// TIA Portal V16 program export: 4 tag tables, 2 data types, 4 data blocks, 31 code blocks (in call order from the OBs), 84 instance data blocks

VAR_GLOBAL   // PLC tag table "Default tag table"
   "Drive 1 Ready" AT %I0.0 : Bool;   // +MC-21K2:1 - Drive 1 Ready
   "Drive 2 Ready" AT %I0.1 : Bool;   // +MC-21K2:5 - Drive 2 Ready
   "Drive 3 Ready" AT %I0.2 : Bool;   // +MC-21K2:2 - Drive 3 Ready
   "Drive 4 Ready" AT %I0.3 : Bool;   // +MC-21K2:6 - Drive 4 Ready
   "Drive 5 Ready" AT %I0.4 : Bool;   // +MC-21K2:3 - Drive 5 Ready
   "Sensor Trechter" AT %I0.5 : Bool;   // +MC-21K2:7 - Sensor Trechter
   "Sensor Op Band" AT %I0.6 : Bool;   // +MC-21K2:4 Sensor Op Band
   "Sensor Wals (Option)" AT %I0.7 : Bool;   // +MC-21K2:8 - Sensor Wals (Option)
   "ESB Oke" AT %I1.0 : Bool;   // +MC-21K3:1 - ESB Oke
   "ESB Pressend" AT %I1.1 : Bool;   // +MC-21K3:5 - ESB Pressend
   "Reset Active" AT %I1.2 : Bool;   // +MC-21K3:2 - Reset Active
   "Noodsleutel(1)" AT %I1.3 : Bool;   // +MC-21K3:6 - NOODSLEUTEL
   "Alle uitgangen(1)" AT %I1.4 : Bool;   // +MC-21K3:3 - Alle uitgangen
   "Door 1 NC contact" AT %I1.5 : Bool;   // +MC-21K3:7 - Safety Doorswitch 1
   "Door 1 NO contact" AT %I1.6 : Bool;   // +MC-21K3:4 - Safety Doorswitch 1 Normaly open
   "Door 2 NC contact" AT %I1.7 : Bool;   // +MC-21K3:8 - Safety Doorswitch 2
   "Spare(5)" AT %I3.0 : Bool;
   "Spare(6)" AT %I3.1 : Bool;
   "Spare(10)" AT %I180.0 : Bool;   // Spare
   "Spare(11)" AT %I180.1 : Bool;   // Spare
   "Spare(12)" AT %I3.4 : Bool;   // Spare
   "Spare(13)" AT %I3.5 : Bool;   // Spare
   "Spare(14)" AT %I3.6 : Bool;   // Spare
   "Spare(15)" AT %I3.7 : Bool;   // Spare
   "Programma 1" AT %I2.0 : Bool;   // +MC-21K4:1 - Programma 1
   "Programma 2" AT %I2.1 : Bool;   // +MC-21K4:5 - Programma 2 (Option)
   "Programma 3" AT %I2.2 : Bool;   // +MC-21K4:2 - Programma 3
   Cleaning AT %I2.3 : Bool;   // +MC-21K4:6 - Cleaning
   "Start Machine" AT %I2.4 : Bool;   // +MC-21K4:3 - Start Machine
   "Stop Machine" AT %I2.5 : Bool;   // +MC-21K4:7 - Stop Machine
   "Spare(16)" AT %I2.6 : Bool;   // Spare
   Encoder_Z_Puls AT %I2.7 : Bool;   // Spare
   "Safety Relais" AT %Q0.0 : Bool;   // +MC-21K6:1 - Safety Relais
   "Bel Storing" AT %Q0.1 : Bool;   // +MC-21K6:5 - Bel Storing
   Spare AT %Q5.3 : Bool;   // Spare
   "Drive 1 RUN FWD" AT %Q1.0 : Bool;   // +MC-21K8:1 - Drive 1 RUN FWD
   "Drive 1 REV]" AT %Q1.1 : Bool;   // +MC-21K8:5 - Drive 1 REV
   "Drive 1 Speed 1" AT %Q1.2 : Bool;   // +MC-21K8:2 - Drive 1 Speed 1
   "Drive 1 Speed 2" AT %Q1.3 : Bool;   // +MC-21K8:6 - Drive 1 Speed 2
   "Spare(3)" AT %Q1.4 : Bool;   // Spare
   "Drive 2 RUN FWD" AT %Q1.5 : Bool;   // +MC-21K8:7 - Drive 2 RUN FWD
   "Drive 2 REV" AT %Q1.6 : Bool;   // +MC-21K8:4 - Drive 2 REV
   "Drive 2 Speed 1" AT %Q1.7 : Bool;   // +MC-21K8:8 - Drive 2 Speed 1
   "Drive 2 Speed 2" AT %Q2.0 : Bool;   // +MC-21K9:1 - Drive 2 Speed 2
   "Spare(4)" AT %Q2.1 : Bool;   // Spare
   "Drive 3 RUN FWD" AT %Q2.2 : Bool;   // +MC-21K9:2 - Drive 3 RUN FWD
   "Drive 3 REV" AT %Q2.3 : Bool;   // +MC-21K9:6 - Drive 3 REV
   "Drive 3 Speed 1" AT %Q2.4 : Bool;   // +MC-21K9:3 - Drive 3 Speed 1
   "Drive 3 Speed 2" AT %Q2.5 : Bool;   // +MC-21K9:7 - Drive 3 Speed 2
   "Spare(21)" AT %Q2.6 : Bool;   // Spare
   "Drive 4 RUN FWD" AT %Q2.7 : Bool;   // +MC-21K9:8 - Drive 4 RUN FWD
   "Drive 4 REV" AT %Q3.0 : Bool;   // +MC-21K10:1 - Drive 4 REV
   "Drive 4 Speed 1" AT %Q3.1 : Bool;   // +MC-21K10:5 - Drive 4 Speed 1
   "Drive 4 Speed 2" AT %Q3.2 : Bool;   // +MC-21K10:2 - Drive 4 Speed 2
   "Spare(22)" AT %Q3.3 : Bool;   // Spare
   "Drive 5 RUN FWD" AT %Q3.4 : Bool;   // +MC-21K10:3 - Drive 5 RUN FWD
   "Drive 5 REV" AT %Q3.5 : Bool;   // +MC-21K10:7 - Drive 5 REV
   "Drive 5 Speed 1" AT %Q3.6 : Bool;   // +MC-21K10:4 - Drive 5 Speed 1
   "Drive 5 Speed 2" AT %Q3.7 : Bool;   // +MC-21K10:8 - Drive 5 Speed 2
   "Spare(23)" AT %Q4.0 : Bool;   // Spare
   "LED Programma 1" AT %Q4.1 : Bool;   // +MC-21K11:5 - LED Programma 1
   "LED Programma 2" AT %Q4.2 : Bool;   // +MC-21K11:2 - LED Programma 2
   "LED Programma 3" AT %Q4.3 : Bool;   // +MC-21K11:6 - LED Programma 3
   "LED E-STOP" AT %Q0.2 : Bool;   // +MC-21K6:2- LED E-STOP
   "LED RUN" AT %Q4.5 : Bool;   // +MC-21K11:7 - LED RUN
   "Valve 1" AT %Q4.6 : Bool;   // +MC-21K11:4 - Valve 1
   "Valve 2" AT %Q4.7 : Bool;   // +MC-21K11:8 - Valve 2
   "Valve 3" AT %Q5.0 : Bool;   // +MC-21K12:1 - Valve 3
   "Valve 4" AT %Q5.1 : Bool;   // +MC-21K12:5 - Valve 4
   "Valve 5" AT %Q5.2 : Bool;   // +MC-21K12:2 - Valve 5
   "Spare(1)" AT %Q6.0 : Bool;   // Spare
   "Spare(2)" AT %Q6.1 : Bool;   // Spare
   "Spare(18)" AT %Q6.2 : Bool;   // Spare
   "Spare(19)" AT %Q6.3 : Bool;   // Spare
   "Spare(20)" AT %Q4.4 : Bool;   // Spare
   "Drive 1 Rapid Stop" AT %Q0.3 : Bool;   // +MC-21K6:6 - Drive 1 Rapid Stop
   "Drive 2 Rapid Stop" AT %Q0.4 : Bool;   // +MC-21K6:3 - Drive 2 Rapid Stop
   "Drive 3 Rapid Stop" AT %Q0.5 : Bool;   // +MC-21K6:7 - Drive 3 Rapid Stop
   "Drive 4 Rapid Stop" AT %Q0.6 : Bool;   // +MC-21K6:4 - Drive 4 Rapid Stop
   "Drive 5 Rapid Stop" AT %Q0.7 : Bool;   // +MC-21K6:8 - Drive 5 Rapid Stop
   "Systeem RUN" AT %M0.0 : Bool;   // Systeem RUN
   Tag_1 AT %M0.1 : Bool;
   Tag_2 AT %M0.2 : Bool;
   Tag_3 AT %M0.3 : Bool;
   Tag_4 AT %M0.4 : Bool;
   "Safety Feedback" AT %M0.6 : Bool;
   Tag_5 AT %M0.7 : Bool;
   Tag_6 AT %M1.0 : Bool;
   "ONC Drive 1 RUN FWD" AT %M10.0 : Bool;
   "ONC Drive 2 RUN FWD" AT %M10.1 : Bool;
   "ONC Drive 3 RUN FWD" AT %M10.2 : Bool;
   "ONC Drive 4 RUN FWD" AT %M10.3 : Bool;
   "ONC Drive 5 RUN FWD" AT %M10.4 : Bool;
   "ONC Drive 1 RUN FWD and Speed 1" AT %M10.5 : Bool;
   "ONC Drive 2 RUN FWD and Speed 1" AT %M10.6 : Bool;
   "ONC Drive 3 RUN FWD and Speed 1" AT %M10.7 : Bool;
   "ONC Drive 4 RUN FWD and Speed 1" AT %M11.0 : Bool;
   "ONC Drive 5 RUN FWD and Speed 1" AT %M11.1 : Bool;
   "ONC Drive 1 RUN FWD and Speed 2" AT %M11.2 : Bool;
   "ONC Drive 2 RUN FWD and Speed 2" AT %M11.3 : Bool;
   "ONC Drive 3 RUN FWD and Speed 2" AT %M11.4 : Bool;
   "ONC Drive 4 RUN FWD and Speed 2" AT %M11.5 : Bool;
   "ONC Drive 5 RUN FWD and Speed 2" AT %M11.6 : Bool;
   Startknop_Scherm AT %M15.0 : Bool;
   Stopknop_Scherm AT %M15.1 : Bool;
   Tag_7 AT %M110.1 : Bool;
   Reset_scherm AT %M15.2 : Bool;
   Sensor_op_band_memory AT %M15.3 : Bool;
   "System RUN_1" AT %M20.0 : Bool;
   ResetDelay AT %M20.1 : Bool;
   SensorWalsMemory AT %M20.2 : Bool;
   Timer_Memory AT %M20.3 : Bool;
   StopAll AT %M20.4 : Bool;
   Tag_8 AT %M100.3 : Bool;
   Tag_9 AT %M100.4 : Bool;
   Tag_10 AT %M0.5 : Bool;
   Tag_11 AT %M150.0 : Bool;
   Tag_12 AT %M101.1 : Bool;
   Tag_13 AT %T1 : Timer;
   Tag_14 AT %M300.0 : Bool;
   Tag_15 AT %M260.0 : Bool;
   Tag_16 AT %M300.1 : Bool;
   Tag_17 AT %M501.0 : Bool;
   Tag_18 AT %M500.1 : Bool;
   Tag_19 AT %M160.0 : Bool;
   Tag_20 AT %M150.5 : Bool;
   Tag_21 AT %QD256 : DWord;
   Tag_22 AT %QW260 : Word;
   Tag_23 AT %ID256 : DWord;
   Tag_24 AT %ID260 : DWord;
   Tag_25 AT %ID464 : DWord;
   Tag_26 AT %ID471 : DWord;
   Tag_27 AT %QW471 : Word;
   Tag_28 AT %QD464 : DWord;
   Tag_30 AT %IW205 : Int;
   SystemTime AT %MD2 : Time;
   Tag_31 AT %M5.0 : Bool;
   Lamp_Green AT %Q7.0 : Bool;
   Lamp_Blue AT %Q7.1 : Bool;
   Lamp_Yellow AT %Q7.2 : Bool;
   Lamp_Red AT %Q7.3 : Bool;
   Lamp_Buzzer AT %Q7.4 : Bool;
   PulseTimer AT %T0 : Timer;
END_VAR

VAR_GLOBAL   // PLC tag table "PositionControl"
   Counter1_IW100 AT %IW100 : Int;
   Counter2_IW102 AT %IW102 : Int;
   "Manual Jog Fwd" AT %M137.0 : Bool;
   "Manual Jog Rev" AT %M137.1 : Bool;
   ReferenceSwitchAxis3 AT %I3.0 : Bool;
   EncoderBand_Alive AT %IW110 : Int;
   EncoderBand_RawCounter AT %IW112 : Int;
   EncoderBand_FineCounter AT %IW113 : Int;
   Zpuls_Encoder_Band AT %I110.3 : Bool;
END_VAR

VAR_GLOBAL   // PLC tag table "Secund. Tags"
   Aanvoerband_Tag1 AT %M100.0 : Bool;
   Aanvoerband_Tag2 AT %M100.1 : Bool;
   Trechter_Bijvullen_Haltveroorzaker AT %M100.2 : Bool;
   Safety_Automatic AT %M100.5 : Bool;
   Safety_Override AT %M100.6 : Bool;
   RUN_Automatic AT %M100.7 : Bool;
   RUN_Manual AT %M101.0 : Bool;
   Invert_Trechter_Sensor AT %M101.2 : Bool;
   WalsSensorMemory AT %M101.3 : Bool;
   Disable_Module AT %M101.4 : Bool;
   Sensor_Trechter_Delayed AT %M101.5 : Bool;
   Positive_Flank AT %M101.6 : Bool;
   ProductSensor_Flank AT %M101.7 : Bool;
   ProductSensor_Rug AT %M102.0 : Bool;
   SensorRug AT %M102.1 : Bool;
   TimeCyclusEnd AT %M102.2 : Bool;
   CounterReset AT %M102.3 : Bool;
   StartTimer AT %M102.4 : Bool;
   StopTimer AT %M102.5 : Bool;
   SaveTimervalue AT %M102.6 : Bool;
   ResetTotalProducts AT %M102.7 : Bool;
   MaintenanceNeeded AT %M103.0 : Bool;
   RetainValues AT %M112.0 : Bool;
   "Retain_1_DontTouch!" AT %M112.1 : Bool;
   Safety_Doors AT %M112.2 : Bool;
   Overname_Linked_Drive1 AT %M112.3 : Bool;
   Drive_RefuseLinkingDrive1 AT %M112.4 : Bool;
   Drive_4_Speed1_Link AT %M112.5 : Bool;
   Drive_4_Speed1_Unlink AT %M112.6 : Bool;
   SafetyOK AT %M112.7 : Bool;
   Valve2_Pulse AT %M113.0 : Bool;
END_VAR

VAR_GLOBAL   // PLC tag table "Tag table_1"
END_VAR

TYPE "ProductEntry"
// stored: IsFailsafeCompliant false
   STRUCT
      StartTime : Time := T#0ms;
      Active : Bool;
   END_STRUCT;
END_TYPE

TYPE "ProductTrack"
// stored: IsFailsafeCompliant false
   STRUCT
      StartPosition : Real;
      Active : Bool;
   END_STRUCT;
END_TYPE

DATA_BLOCK "PLCMemory"   // DB15
VERSION : 0.1
// stored: AutoNumber true, IsOnlyStoredInLoadMemory false, IsWriteProtectedInAS false
   VAR RETAIN
      Homing_Sensor_Wals_Offset_Test : Time := T#1S_200MS;   // Offset of homing position sensor wals
      Wals_Delay_Offset : Time := T#400MS;   // Offset of Wals on delay
      Safety_Delay : Time := T#5MS;   // Delay of safety high
      WalsCheck_Time : Time := T#5S;   // Time offset when wals slipping message is displayed
      ProductCheck_Time : Time := T#15S;   // Time offset when aanvoer not in position message is displayed
      ProductIntervalTime : Time;   // Counts the time between 2 products
      ProductIntervalTime_1 : Time;   // Depends on ProductIntervalTimer
      ProductIntervalTime_2 : Time;   // Depends on ProductIntervalTimer_1
      TD_Products_Counter : Int;   // Counts the total amount of products with the Sensor Band
      UsernameMemory : String := 'Key';
      PasswordMemory : String := 'Key123';
      SpeedSettingsTakeover : Bool := True;   // Makes the speed of Overname the same as speed Drive 1
      SpeedSettingOvername : Bool;   // Parameter of setting the speed for Drive 4 (Overname)
      SpeedSettingBand : Bool;   // Parameter of setting the speed for Drive 1 (Band)
      TimingSettingOvername : Bool := True;   // Makes the timing of Overname the same as speed Drive 1
      EncoderPosition : Real;   // Real Value of Encoder Axis 3 (Wals)
      StepSize : Real := 0.0;   // Pulsfactor of Encoder Axis 3
      Desired_Encoder_Position : Real;
      Tolerance : Real := 0.0;
      "Encoder PulsOffset" : Time := T#3MS;
      Axis3_Ref_Pos : Real := 85.0;   // Refention position of Axis 3 without tolerance
      Reference_Position_Axis3 : Real;   // Refention position of Axis 3 with calculated tolerance
      ProductCount : Int;
      Axis3_ControlMode : Bool := true;
      Axis1_ControlMode : Bool := true;
      ProductsToProduce : Int;
      SystemTime : Time;
      Disable_Modules : Struct
         Disable_Band : Bool;
         Disable_Trilgoten : Bool;
         Disable_AanvoerWals : Bool;
         Disable_Aandruk1 : Bool;
         Disable_Aandruk2 : Bool;
         Disable_Aandruk3 : Bool;
         Disable_Blaaspuls : Bool;
         Disable_Retourband : Bool;
         Disable_Afsluiter : Bool;
      END_STRUCT;
      Offset_Timers : Struct
         Trilgoten_Start_Offset : Time := T#10MS;   // Delay offset of start trilgoten
         Trilgoten_Stop_Offset : Time := T#10MS;   // Delay offset of stop trilgoten
         Aanvoer_Start_Offset : Time := T#10MS;   // Delay offset of start aanvoer
         Magazijn_Sensor_Delay : Time := T#15S;   // Delay on magazijn sensor.
         Aanvoer_Stop_Offset : Time := T#10MS;   // Delay offset of stop aanvoer
         Overname_Start_Offset : Time := T#5MS;   // Delay offset of start Overname
         Overname_Stop_Offset : Time := T#5MS;   // Delay offset of stop Overname
         Retourband_Start_Offset : Time := T#5ms;
         Retourband_Stop_Offset : Time := T#5ms;
         BlowOff_CycleTime : Time := T#500ms;
         Blow_Off_PulseTime : Time := T#500ms;
      END_STRUCT;
      ProductBuffer : Struct
         DelayTime : Time := T#7s;
         ProductsCount : Int;
         MoveTrigger : Bool;
         MoveFeedback : Bool;
         RestFeedback : Bool;
         InsertIndex : Int;
      END_STRUCT;
      ProductBufferBehindWals : Struct
         DelayTime : Time := T#2s_500MS;
         Product_Count : Int;
      END_STRUCT;
   END_VAR
BEGIN
END_DATA_BLOCK

DATA_BLOCK "DB_SystemTimeCounter"   // DB68
VERSION : 0.1
// stored: AutoNumber true, IsOnlyStoredInLoadMemory false, IsWriteProtectedInAS false
   VAR RETAIN
      SystemTime : Time;
   END_VAR
BEGIN
END_DATA_BLOCK

DATA_BLOCK "Alarms"   // DB24
VERSION : 0.1
// stored: AutoNumber true, IsOnlyStoredInLoadMemory false, IsWriteProtectedInAS false
   VAR
      AlarmStruct : Struct
         Alarm_Product_Not_Position : Bool;
         Alarm_Axis_Not_Position : Bool;
         Alarm_Drive1 : Bool;
         Alarm_Drive2 : Bool;
         Alarm_Drive3 : Bool;
         Alarm_Drive4 : Bool;
         Alarm_Drive5 : Bool;
         "Alarm_To_Many_Products_Reset_Counter!" : Bool;
      END_STRUCT;
      AlarmsWord : Word;
      HMI_Alarm_Drive1 : Word;
      HMI_Alarm_Drive2 : Word;
      HMI_Alarm_Drive3 : Word;
      HMI_Alarm_Drive4 : Word;
      HMI_Alarm_Drive5 : Word;
   END_VAR
BEGIN
END_DATA_BLOCK

DATA_BLOCK "PositionManagement"   // DB51
VERSION : 0.1
// stored: AutoNumber true, IsOnlyStoredInLoadMemory false, IsWriteProtectedInAS false
   VAR RETAIN
      Data : Struct   // Data
         CntPlsPrev : DInt := 0;   // Flowpulsen vorige scan
         CntPlsDiff : DInt := 0;   // Flowpulsen verschil
         CntPlsAct : DInt := 0;   // Flowpulsen actueel
         DosActueel : Real := 0.0;   // Dosering actueel ('x' gram/liter/kg gist)
         Actual_Axis3_Position : Real;   // Actual Position of Axis 3 stored in this datablock
         Actual_Axis1_Position : Real;
      END_STRUCT;
      "Axis 3" : Struct
         Values : Struct
            AxisName : String := 'Drive 3 - Wals';
            "Reference Position" : Int := 0;
            "Set Position" : Real := -50.0;
            "Rest Position" : Real := -25.0;
            Acceleration : Real := 0.0;
            Deacceleration : Real;
            "Axis Correction" : Real := 1.0E-06;
            "Position Offset" : Real := 35.0;
            Pulsfactor : Real := 0.82;
            Axis_Speed : Int := 0;
         END_STRUCT;
         Commands : Struct
            "Go To Rest" : Bool;
            "Start Ref Run" : Bool;
            "Take Over Pos" : Bool;
            "Go To Position" : Bool;
            "Jog Fwd" : Bool;
            "Jog Rev" : Bool;
            Axis_Brake : Bool;
            MasterWord : String;
            "Master Callback" : String;
         END_STRUCT;
         Messages : Struct
            "Axis Busy" : Bool;
            "Error Executing Command" : Bool;
            "Axis On Rest" : Bool;
            "Axis On Position" : Bool;
            "Drive State (Option)" : String;
            "Slip State" : String;
            AxisHasReference : Bool;
         END_STRUCT;
      END_STRUCT;
      Demo_Pos : Struct
         Desired_Pos : Real;
         Start : Bool;
         SetRefRunActive : Bool;
         RequestMove1 : Bool;
         RequestMove2 : Bool;
         PositionMove2 : Real := -330.0;
         PositionMove1 : Real := -120.0;
         Pos2Done : Bool;
         BrakeOnPos1 : Bool;
         BrakeOnPos2 : Bool;
         ManualSensorOverride : Bool;
      END_STRUCT;
      Axis_1 : Struct
         Values : Struct
            AxisName : String := 'Drive 1 - Infeed';
            "Reference Position" : Int := 0;
            "Set Position" : Real := 0.0;
            "Rest Position" : Real := 0.0;
            Acceleration : Real := 0.0;
            Deacceleration : Real;
            "Axis Correction" : Real := 1.0E-06;
            "Position Offset" : Real := 0.001;
            Pulsfactor : Real := -0.325;
            Axis_Speed : Int := 0;
         END_STRUCT;
         Commands : Struct
            "Go To Rest" : Bool;
            "Start Ref Run" : Bool;
            "Take Over Pos" : Bool;
            "Go To Position" : Bool;
            "Jog Fwd" : Bool;
            "Jog Rev" : Bool;
            Axis_Brake : Bool;
            ReferenceSwitch : Bool;
            MasterWord : String;
            "Master Callback" : String;
         END_STRUCT;
         Messages : Struct
            "Axis Busy" : Bool;
            "Error Executing Command" : Bool;
            "Axis On Rest" : Bool;
            "Axis On Position" : Bool;
            "Drive State (Option)" : String;
            "Slip State" : String;
            AxisHasReference : Bool;
         END_STRUCT;
      END_STRUCT;
   END_VAR
BEGIN
END_DATA_BLOCK

ORGANIZATION_BLOCK "OB1"   // OB1, LAD, ProgramCycle
TITLE = MAIN Program
VERSION : 0.1
// MAIN Block
// stored: IsIECCheckEnabled false
   VAR_TEMP
      Temp_0 : Byte;
      Temp_1 : Byte;
      Temp_2 : Byte;
      Temp_3 : Byte;
      Temp_4 : Byte;
      Temp_5 : Byte;
      Temp_6 : Int;
      Temp_7 : Int;
      Temp_8 : Int;
      Temp_9 : Date_And_Time;
      Temp_10 : DWord;
      EncoderDirection : Bool;
      HomingActive : Bool;
      EncError : Bool;
      SafetyActive : Bool;
      "Spare Drive 6" : Bool;
      "Spare Drive 7" : Bool;
      "Spare Drive 8" : Bool;
      "Spare Drive 9" : Bool;
      "Spare Drive 10" : Bool;
      SAFE_OK_Signal : Bool;
      Raw_Position : Real;
      Encoder : Int;
      Gate : Bool;
      GATESTP : Bool;
      OTERRA : Bool;
      Direct : Bool;
      Prepar : Bool;
      CMPV1 : Bool;
      CMPV2 : Bool;
      RESSYNC : Bool;
      RESZERO : Bool;
      OTERR : Bool;
      UnscPos : Int;
      Sc_Pos : Int;
      ActEncPos : Real;
      Start_ReferenceRun : Bool;
      ReferenceSwitch_Input : Bool;
      "Reference Position" : Real;
      "Jog FWD" : Bool;
      "Jog REV" : Bool;
      RefSwitchTemp : Bool;
      RefPosDint : DInt;
      RefPosInt : Real;
      Start_Movement : Bool;
      ClockTime : Int;
      LT_Time : Date_And_Time;
      Summer : Bool;
      SystemStartUp : Bool;
      StartupLow : Bool;
      ManualSensorOverride : Bool;
      Axis1_ScaledPosition : Real;
      Axis1_ActualEncPosition : Real;
   END_VAR
   VAR_TEMP   // added for the SCL form of the ladder/FBD networks
      _w1 : Bool;
   END_VAR
BEGIN

REGION Network 1: Retain Variables
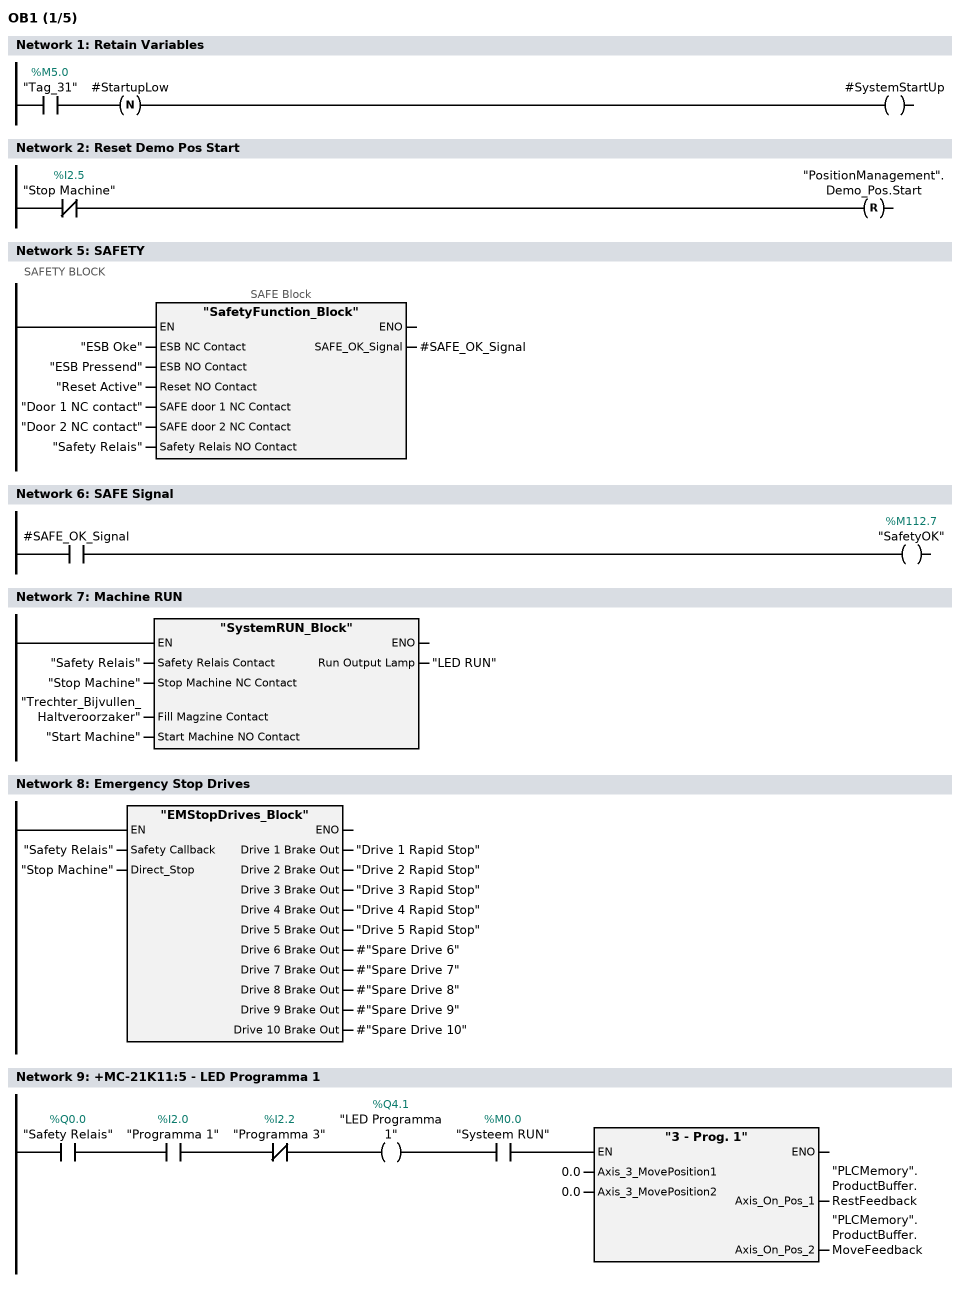
   RUNG wire#powerrail
      Contact( "Tag_31" )
      N_Trig( #StartupLow )
      Coil( #SystemStartUp )
   END_RUNG
   // the same network as SCL:
   #_w1 := NOT "Tag_31" AND #StartupLow;   // falling edge
   #StartupLow := "Tag_31";
   #SystemStartUp := #_w1;
END_REGION

REGION Network 2: Reset Demo Pos Start
   RUNG wire#powerrail
      I_Contact( "Stop Machine" )
      R_Coil( "PositionManagement".Demo_Pos.Start )
   END_RUNG
   // the same network as SCL:
   IF NOT "Stop Machine" THEN "PositionManagement".Demo_Pos.Start := FALSE; END_IF;
END_REGION

REGION Network 3: Retain Veriables (2)
END_REGION

REGION Network 4: System Time
END_REGION

REGION Network 5: SAFETY
   // SAFETY BLOCK
   RUNG wire#powerrail
      "SafetyFunction_Block"("ESB NC Contact" := "ESB Oke", "ESB NO Contact" := "ESB Pressend", "Reset NO Contact" := "Reset Active", "SAFE door 1 NC Contact" := "Door 1 NC contact", "SAFE door 2 NC Contact" := "Door 2 NC contact", "Safety Relais NO Contact" := "Safety Relais", SAFE_OK_Signal => #SAFE_OK_Signal)   // SAFE Block
   END_RUNG
   // the same network as SCL:
   "SafetyFunction_Block"("ESB NC Contact" := "ESB Oke",   // SAFE Block
                          "ESB NO Contact" := "ESB Pressend",
                          "Reset NO Contact" := "Reset Active",
                          "SAFE door 1 NC Contact" := "Door 1 NC contact",
                          "SAFE door 2 NC Contact" := "Door 2 NC contact",
                          "Safety Relais NO Contact" := "Safety Relais",
                          SAFE_OK_Signal => #SAFE_OK_Signal);
END_REGION

REGION Network 6: SAFE Signal
   RUNG wire#powerrail
      Contact( #SAFE_OK_Signal )
      Coil( "SafetyOK" )
   END_RUNG
   // the same network as SCL:
   "SafetyOK" := #SAFE_OK_Signal;
END_REGION

REGION Network 7: Machine RUN
   RUNG wire#powerrail
      "SystemRUN_Block"("Safety Relais Contact" := "Safety Relais", "Stop Machine NC Contact" := "Stop Machine", "Fill Magzine Contact" := "Trechter_Bijvullen_Haltveroorzaker", "Start Machine NO Contact" := "Start Machine", "Run Output Lamp" => "LED RUN")
   END_RUNG
   // the same network as SCL:
   "SystemRUN_Block"("Safety Relais Contact" := "Safety Relais",
                     "Stop Machine NC Contact" := "Stop Machine",
                     "Fill Magzine Contact" := "Trechter_Bijvullen_Haltveroorzaker",
                     "Start Machine NO Contact" := "Start Machine",
                     "Run Output Lamp" => "LED RUN");
END_REGION

REGION Network 8: Emergency Stop Drives
   RUNG wire#powerrail
      "EMStopDrives_Block"("Safety Callback" := "Safety Relais", Direct_Stop := "Stop Machine", "Drive 1 Brake Out" => "Drive 1 Rapid Stop", "Drive 2 Brake Out" => "Drive 2 Rapid Stop", "Drive 3 Brake Out" => "Drive 3 Rapid Stop", "Drive 4 Brake Out" => "Drive 4 Rapid Stop", "Drive 5 Brake Out" => "Drive 5 Rapid Stop", "Drive 6 Brake Out" => #"Spare Drive 6", "Drive 7 Brake Out" => #"Spare Drive 7", "Drive 8 Brake Out" => #"Spare Drive 8", "Drive 9 Brake Out" => #"Spare Drive 9", "Drive 10 Brake Out" => #"Spare Drive 10")
   END_RUNG
   // the same network as SCL:
   "EMStopDrives_Block"("Safety Callback" := "Safety Relais",
                        Direct_Stop := "Stop Machine",
                        "Drive 1 Brake Out" => "Drive 1 Rapid Stop",
                        "Drive 2 Brake Out" => "Drive 2 Rapid Stop",
                        "Drive 3 Brake Out" => "Drive 3 Rapid Stop",
                        "Drive 4 Brake Out" => "Drive 4 Rapid Stop",
                        "Drive 5 Brake Out" => "Drive 5 Rapid Stop",
                        "Drive 6 Brake Out" => #"Spare Drive 6",
                        "Drive 7 Brake Out" => #"Spare Drive 7",
                        "Drive 8 Brake Out" => #"Spare Drive 8",
                        "Drive 9 Brake Out" => #"Spare Drive 9",
                        "Drive 10 Brake Out" => #"Spare Drive 10");
END_REGION

REGION Network 9: +MC-21K11:5 - LED Programma 1
   RUNG wire#powerrail
      Contact( "Safety Relais" )
      Contact( "Programma 1" )
      I_Contact( "Programma 3" )
      Coil( "LED Programma 1" )
      Contact( "Systeem RUN" )
      "3 - Prog. 1"(Axis_3_MovePosition1 := 0.0, Axis_3_MovePosition2 := 0.0, Axis_On_Pos_1 => "PLCMemory".ProductBuffer.RestFeedback, Axis_On_Pos_2 => "PLCMemory".ProductBuffer.MoveFeedback)
   END_RUNG
   // the same network as SCL:
   "LED Programma 1" := "Safety Relais" AND "Programma 1" AND NOT "Programma 3";
   IF "LED Programma 1" AND "Systeem RUN" THEN
       "3 - Prog. 1"(Axis_3_MovePosition1 := 0.0,
                     Axis_3_MovePosition2 := 0.0,
                     Axis_On_Pos_1 => "PLCMemory".ProductBuffer.RestFeedback,
                     Axis_On_Pos_2 => "PLCMemory".ProductBuffer.MoveFeedback);
   END_IF;
END_REGION

REGION Network 10: +MC-21K11:2 - LED Programma 2
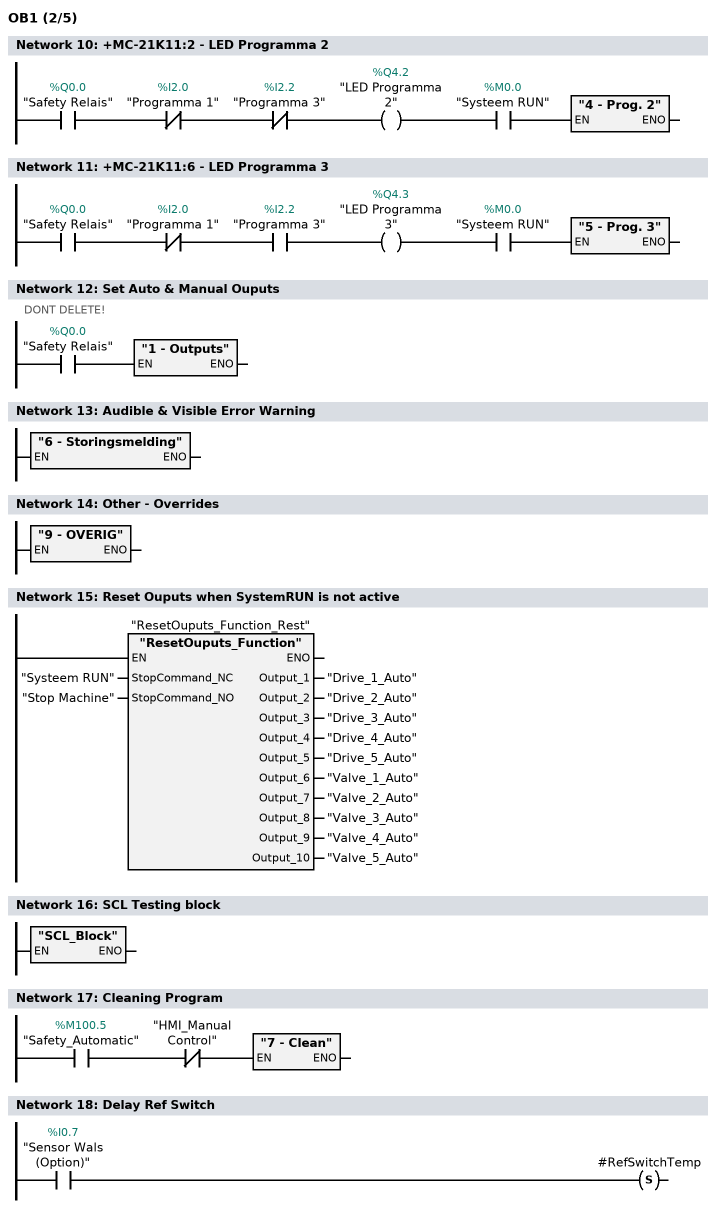
   RUNG wire#powerrail
      Contact( "Safety Relais" )
      I_Contact( "Programma 1" )
      I_Contact( "Programma 3" )
      Coil( "LED Programma 2" )
      Contact( "Systeem RUN" )
      "4 - Prog. 2"()
   END_RUNG
   // the same network as SCL:
   "LED Programma 2" := "Safety Relais" AND NOT "Programma 1" AND NOT "Programma 3";
   IF "LED Programma 2" AND "Systeem RUN" THEN "4 - Prog. 2"(); END_IF;
END_REGION

REGION Network 11: +MC-21K11:6 - LED Programma 3
   RUNG wire#powerrail
      Contact( "Safety Relais" )
      I_Contact( "Programma 1" )
      Contact( "Programma 3" )
      Coil( "LED Programma 3" )
      Contact( "Systeem RUN" )
      "5 - Prog. 3"()
   END_RUNG
   // the same network as SCL:
   "LED Programma 3" := "Safety Relais" AND NOT "Programma 1" AND "Programma 3";
   IF "LED Programma 3" AND "Systeem RUN" THEN "5 - Prog. 3"(); END_IF;
END_REGION

REGION Network 12: Set Auto & Manual Ouputs
   // DONT DELETE!
   RUNG wire#powerrail
      Contact( "Safety Relais" )
      "1 - Outputs"()
   END_RUNG
   // the same network as SCL:
   IF "Safety Relais" THEN "1 - Outputs"(); END_IF;
END_REGION

REGION Network 13: Audible & Visible Error Warning
   RUNG wire#powerrail
      "6 - Storingsmelding"()
   END_RUNG
   // the same network as SCL:
   "6 - Storingsmelding"();
END_REGION

REGION Network 14: Other - Overrides
   RUNG wire#powerrail
      "9 - OVERIG"()
   END_RUNG
   // the same network as SCL:
   "9 - OVERIG"();
END_REGION

REGION Network 15: Reset Ouputs when SystemRUN is not active
   RUNG wire#powerrail
      "ResetOuputs_Function_Rest"(StopCommand_NC := "Systeem RUN", StopCommand_NO := "Stop Machine", Output_1 => "Drive_1_Auto", Output_2 => "Drive_2_Auto", Output_3 => "Drive_3_Auto", Output_4 => "Drive_4_Auto", Output_5 => "Drive_5_Auto", Output_6 => "Valve_1_Auto", Output_7 => "Valve_2_Auto", Output_8 => "Valve_3_Auto", Output_9 => "Valve_4_Auto", Output_10 => "Valve_5_Auto")
   END_RUNG
   // the same network as SCL:
   "ResetOuputs_Function_Rest"(StopCommand_NC := "Systeem RUN",   // "ResetOuputs_Function"
                           StopCommand_NO := "Stop Machine",
                           Output_1 => "Drive_1_Auto",
                           Output_2 => "Drive_2_Auto",
                           Output_3 => "Drive_3_Auto",
                           Output_4 => "Drive_4_Auto",
                           Output_5 => "Drive_5_Auto",
                           Output_6 => "Valve_1_Auto",
                           Output_7 => "Valve_2_Auto",
                           Output_8 => "Valve_3_Auto",
                           Output_9 => "Valve_4_Auto",
                           Output_10 => "Valve_5_Auto");
END_REGION

REGION Network 16: SCL Testing block
   RUNG wire#powerrail
      "SCL_Block"()
   END_RUNG
   // the same network as SCL:
   "SCL_Block"();
END_REGION

REGION Network 17: Cleaning Program
   RUNG wire#powerrail
      Contact( "Safety_Automatic" )
      I_Contact( "HMI_ManualControl" )
      "7 - Clean"()
   END_RUNG
   // the same network as SCL:
   IF "Safety_Automatic" AND NOT "HMI_ManualControl" THEN "7 - Clean"(); END_IF;
END_REGION

REGION Network 18: Delay Ref Switch
   RUNG wire#powerrail
      Contact( "Sensor Wals (Option)" )
      S_Coil( #RefSwitchTemp )
   END_RUNG
   // the same network as SCL:
   IF "Sensor Wals (Option)" THEN #RefSwitchTemp := TRUE; END_IF;
END_REGION

REGION Network 19: Reset Ref Switch Temp
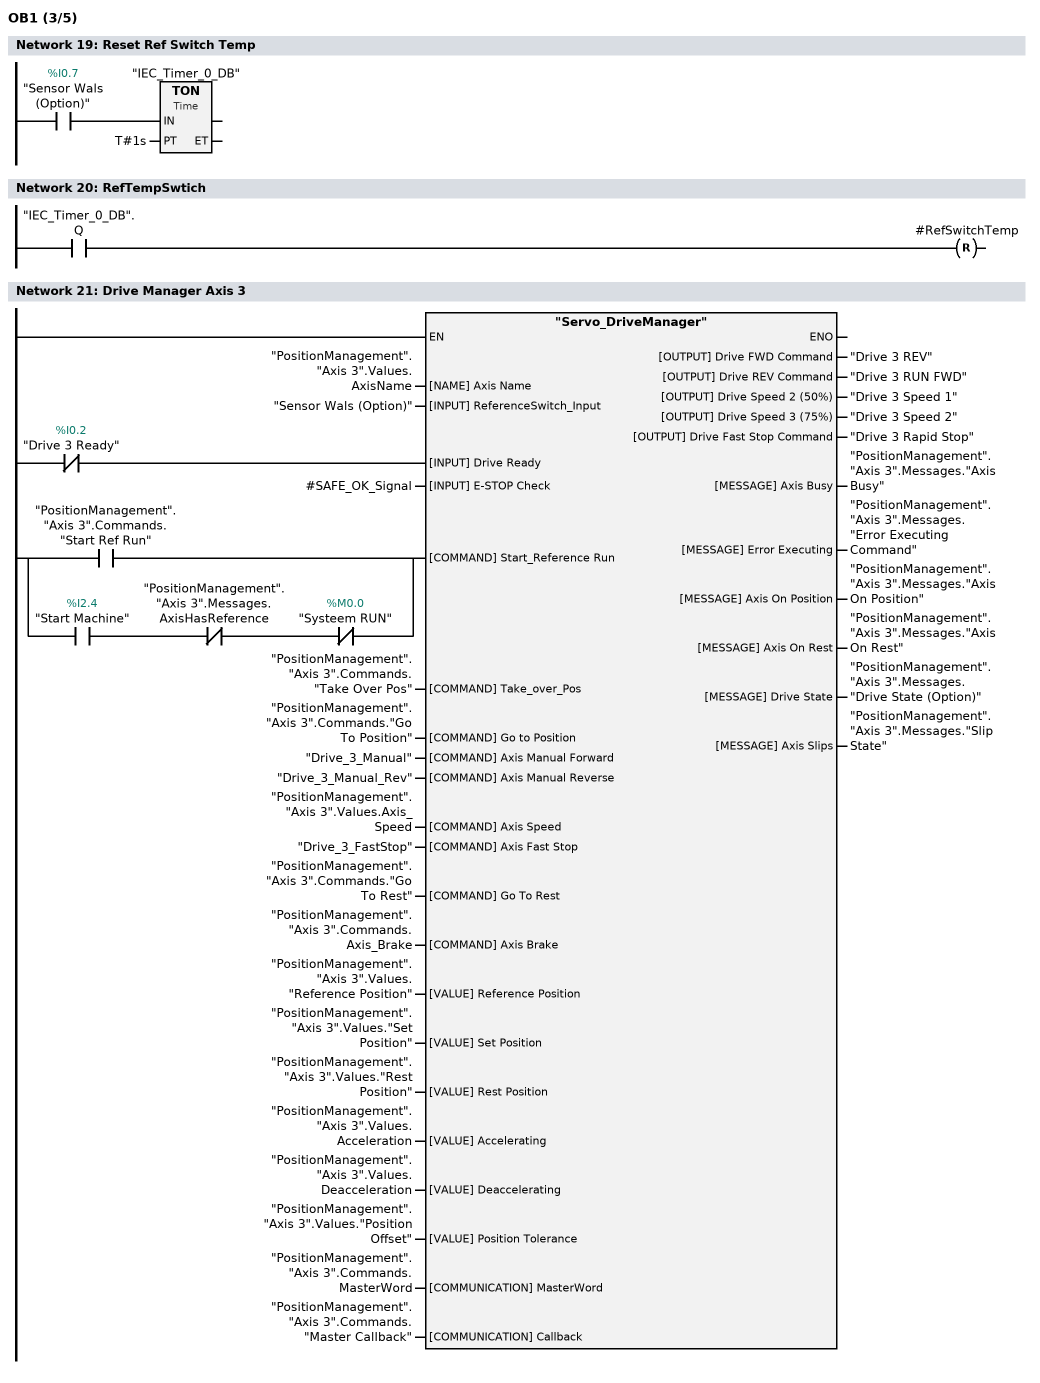
   RUNG wire#powerrail
      Contact( "Sensor Wals (Option)" )
      { S7_Templates := "time_type := Time" } "IEC_Timer_0_DB".TON(pt := T#1s, et =>)
   END_RUNG
   // the same network as SCL:
   "IEC_Timer_0_DB".TON(IN := "Sensor Wals (Option)", PT := T#1s);
END_REGION

REGION Network 20: RefTempSwtich
   RUNG wire#powerrail
      Contact( "IEC_Timer_0_DB".Q )
      R_Coil( #RefSwitchTemp )
   END_RUNG
   // the same network as SCL:
   IF "IEC_Timer_0_DB".Q THEN #RefSwitchTemp := FALSE; END_IF;
END_REGION

REGION Network 21: Drive Manager Axis 3
   RUNG wire#powerrail
      "Servo_DriveManager"("[INPUT] Drive Ready" := wire#w1, "[COMMAND] Start_Reference Run" := wire#w2, "[NAME] Axis Name" := "PositionManagement"."Axis 3".Values.AxisName, "[INPUT] ReferenceSwitch_Input" := "Sensor Wals (Option)", "[INPUT] E-STOP Check" := #SAFE_OK_Signal, "[COMMAND] Take_over_Pos" := "PositionManagement"."Axis 3".Commands."Take Over Pos", "[COMMAND] Go to Position" := "PositionManagement"."Axis 3".Commands."Go To Position", "[COMMAND] Axis Manual Forward" := "Drive_3_Manual", "[COMMAND] Axis Manual Reverse" := "Drive_3_Manual_Rev", "[COMMAND] Axis Speed" := "PositionManagement"."Axis 3".Values.Axis_Speed, "[COMMAND] Axis Fast Stop" := "Drive_3_FastStop", "[COMMAND] Go To Rest" := "PositionManagement"."Axis 3".Commands."Go To Rest", "[COMMAND] Axis Brake" := "PositionManagement"."Axis 3".Commands.Axis_Brake, "[VALUE] Reference Position" := "PositionManagement"."Axis 3".Values."Reference Position", "[VALUE] Set Position" := "PositionManagement"."Axis 3".Values."Set Position", "[VALUE] Rest Position" := "PositionManagement"."Axis 3".Values."Rest Position", "[VALUE] Accelerating" := "PositionManagement"."Axis 3".Values.Acceleration, "[VALUE] Deaccelerating" := "PositionManagement"."Axis 3".Values.Deacceleration, "[VALUE] Position Tolerance" := "PositionManagement"."Axis 3".Values."Position Offset", "[COMMUNICATION] MasterWord" := "PositionManagement"."Axis 3".Commands.MasterWord, "[COMMUNICATION] Callback" := "PositionManagement"."Axis 3".Commands."Master Callback", "[OUTPUT] Drive FWD Command" => "Drive 3 REV", "[OUTPUT] Drive REV Command" => "Drive 3 RUN FWD", "[OUTPUT] Drive Speed 2 (50%)" => "Drive 3 Speed 1", "[OUTPUT] Drive Speed 3 (75%)" => "Drive 3 Speed 2", "[OUTPUT] Drive Fast Stop Command" => "Drive 3 Rapid Stop", "[MESSAGE] Axis Busy" => "PositionManagement"."Axis 3".Messages."Axis Busy", "[MESSAGE] Error Executing" => "PositionManagement"."Axis 3".Messages."Error Executing Command", "[MESSAGE] Axis On Position" => "PositionManagement"."Axis 3".Messages."Axis On Position", "[MESSAGE] Axis On Rest" => "PositionManagement"."Axis 3".Messages."Axis On Rest", "[MESSAGE] Drive State" => "PositionManagement"."Axis 3".Messages."Drive State (Option)", "[MESSAGE] Axis Slips" => "PositionManagement"."Axis 3".Messages."Slip State")
   END_RUNG
   RUNG wire#powerrail
      I_Contact( "Drive 3 Ready" )
   END_RUNG wire#w1
   RUNG wire#powerrail
      Contact( "PositionManagement"."Axis 3".Commands."Start Ref Run" )
   END_RUNG wire#w2
   RUNG wire#powerrail
      Contact( "Start Machine" )
      I_Contact( "PositionManagement"."Axis 3".Messages.AxisHasReference )
      I_Contact( "Systeem RUN" )
   END_RUNG wire#w2
   // the same network as SCL:
   "Servo_DriveManager"("[NAME] Axis Name" := "PositionManagement"."Axis 3".Values.AxisName,
                        "[INPUT] ReferenceSwitch_Input" := "Sensor Wals (Option)",
                        "[INPUT] Drive Ready" := NOT "Drive 3 Ready",
                        "[INPUT] E-STOP Check" := #SAFE_OK_Signal,
                        "[COMMAND] Start_Reference Run" := "PositionManagement"."Axis 3".Commands."Start Ref Run" OR ("Start Machine" AND NOT "PositionManagement"."Axis 3".Messages.AxisHasReference AND NOT "Systeem RUN"),
                        "[COMMAND] Take_over_Pos" := "PositionManagement"."Axis 3".Commands."Take Over Pos",
                        "[COMMAND] Go to Position" := "PositionManagement"."Axis 3".Commands."Go To Position",
                        "[COMMAND] Axis Manual Forward" := "Drive_3_Manual",
                        "[COMMAND] Axis Manual Reverse" := "Drive_3_Manual_Rev",
                        "[COMMAND] Axis Speed" := "PositionManagement"."Axis 3".Values.Axis_Speed,
                        "[COMMAND] Axis Fast Stop" := "Drive_3_FastStop",
                        "[COMMAND] Go To Rest" := "PositionManagement"."Axis 3".Commands."Go To Rest",
                        "[COMMAND] Axis Brake" := "PositionManagement"."Axis 3".Commands.Axis_Brake,
                        "[VALUE] Reference Position" := "PositionManagement"."Axis 3".Values."Reference Position",
                        "[VALUE] Set Position" := "PositionManagement"."Axis 3".Values."Set Position",
                        "[VALUE] Rest Position" := "PositionManagement"."Axis 3".Values."Rest Position",
                        "[VALUE] Accelerating" := "PositionManagement"."Axis 3".Values.Acceleration,
                        "[VALUE] Deaccelerating" := "PositionManagement"."Axis 3".Values.Deacceleration,
                        "[VALUE] Position Tolerance" := "PositionManagement"."Axis 3".Values."Position Offset",
                        "[COMMUNICATION] MasterWord" := "PositionManagement"."Axis 3".Commands.MasterWord,
                        "[COMMUNICATION] Callback" := "PositionManagement"."Axis 3".Commands."Master Callback",
                        "[OUTPUT] Drive FWD Command" => "Drive 3 REV",
                        "[OUTPUT] Drive REV Command" => "Drive 3 RUN FWD",
                        "[OUTPUT] Drive Speed 2 (50%)" => "Drive 3 Speed 1",
                        "[OUTPUT] Drive Speed 3 (75%)" => "Drive 3 Speed 2",
                        "[OUTPUT] Drive Fast Stop Command" => "Drive 3 Rapid Stop",
                        "[MESSAGE] Axis Busy" => "PositionManagement"."Axis 3".Messages."Axis Busy",
                        "[MESSAGE] Error Executing" => "PositionManagement"."Axis 3".Messages."Error Executing Command",
                        "[MESSAGE] Axis On Position" => "PositionManagement"."Axis 3".Messages."Axis On Position",
                        "[MESSAGE] Axis On Rest" => "PositionManagement"."Axis 3".Messages."Axis On Rest",
                        "[MESSAGE] Drive State" => "PositionManagement"."Axis 3".Messages."Drive State (Option)",
                        "[MESSAGE] Axis Slips" => "PositionManagement"."Axis 3".Messages."Slip State");
END_REGION

REGION Network 22: Noodsleutel
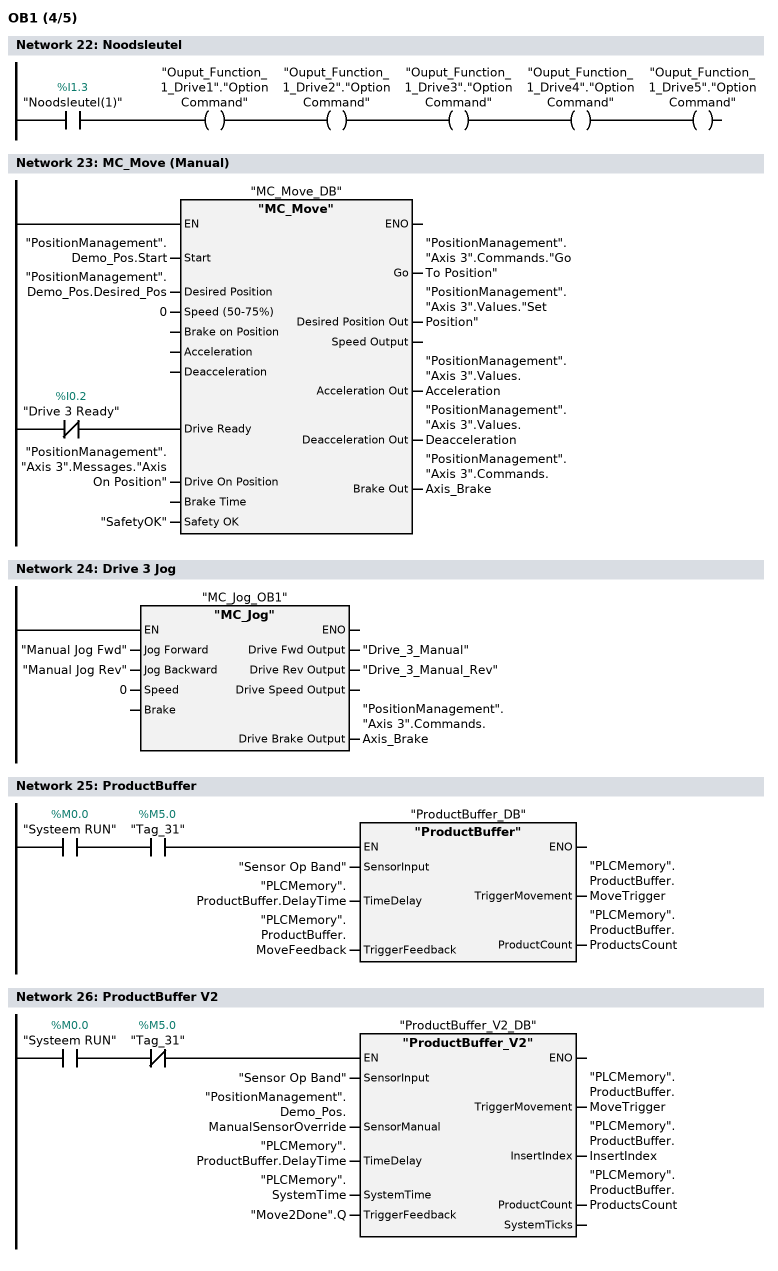
   RUNG wire#powerrail
      Contact( "Noodsleutel(1)" )
      Coil( "Ouput_Function_1_Drive1"."Option Command" )
      Coil( "Ouput_Function_1_Drive2"."Option Command" )
      Coil( "Ouput_Function_1_Drive3"."Option Command" )
      Coil( "Ouput_Function_1_Drive4"."Option Command" )
      Coil( "Ouput_Function_1_Drive5"."Option Command" )
   END_RUNG
   // the same network as SCL:
   "Ouput_Function_1_Drive1"."Option Command" := "Noodsleutel(1)";
   "Ouput_Function_1_Drive2"."Option Command" := "Noodsleutel(1)";
   "Ouput_Function_1_Drive3"."Option Command" := "Noodsleutel(1)";
   "Ouput_Function_1_Drive4"."Option Command" := "Noodsleutel(1)";
   "Ouput_Function_1_Drive5"."Option Command" := "Noodsleutel(1)";
END_REGION

REGION Network 23: MC_Move (Manual)
   RUNG wire#powerrail
      "MC_Move_DB"("Drive Ready" := wire#w1, Start := "PositionManagement".Demo_Pos.Start, "Desired Position" := "PositionManagement".Demo_Pos.Desired_Pos, "Speed (50-75%)" := 0, "Brake on Position" :=, Acceleration :=, Deacceleration :=, "Drive On Position" := "PositionManagement"."Axis 3".Messages."Axis On Position", "Brake Time" :=, "Safety OK" := "SafetyOK", Go => "PositionManagement"."Axis 3".Commands."Go To Position", "Desired Position Out" => "PositionManagement"."Axis 3".Values."Set Position", "Speed Output" =>, "Acceleration Out" => "PositionManagement"."Axis 3".Values.Acceleration, "Deacceleration Out" => "PositionManagement"."Axis 3".Values.Deacceleration, "Brake Out" => "PositionManagement"."Axis 3".Commands.Axis_Brake)
   END_RUNG
   RUNG wire#powerrail
      I_Contact( "Drive 3 Ready" )
   END_RUNG wire#w1
   // the same network as SCL:
   "MC_Move_DB"(Start := "PositionManagement".Demo_Pos.Start,   // "MC_Move"
                "Desired Position" := "PositionManagement".Demo_Pos.Desired_Pos,
                "Speed (50-75%)" := 0,
                "Drive Ready" := NOT "Drive 3 Ready",
                "Drive On Position" := "PositionManagement"."Axis 3".Messages."Axis On Position",
                "Safety OK" := "SafetyOK",
                Go => "PositionManagement"."Axis 3".Commands."Go To Position",
                "Desired Position Out" => "PositionManagement"."Axis 3".Values."Set Position",
                "Acceleration Out" => "PositionManagement"."Axis 3".Values.Acceleration,
                "Deacceleration Out" => "PositionManagement"."Axis 3".Values.Deacceleration,
                "Brake Out" => "PositionManagement"."Axis 3".Commands.Axis_Brake);
END_REGION

REGION Network 24: Drive 3 Jog
   RUNG wire#powerrail
      "MC_Jog_OB1"("Jog Forward" := "Manual Jog Fwd", "Jog Backward" := "Manual Jog Rev", Speed := 0, Brake :=, "Drive Fwd Output" => "Drive_3_Manual", "Drive Rev Output" => "Drive_3_Manual_Rev", "Drive Speed Output" =>, "Drive Brake Output" => "PositionManagement"."Axis 3".Commands.Axis_Brake)
   END_RUNG
   // the same network as SCL:
   "MC_Jog_OB1"("Jog Forward" := "Manual Jog Fwd",   // "MC_Jog"
                "Jog Backward" := "Manual Jog Rev",
                Speed := 0,
                "Drive Fwd Output" => "Drive_3_Manual",
                "Drive Rev Output" => "Drive_3_Manual_Rev",
                "Drive Brake Output" => "PositionManagement"."Axis 3".Commands.Axis_Brake);
END_REGION

REGION Network 25: ProductBuffer
   RUNG wire#powerrail
      Contact( "Systeem RUN" )
      Contact( "Tag_31" )
      "ProductBuffer_DB"(SensorInput := "Sensor Op Band", TimeDelay := "PLCMemory".ProductBuffer.DelayTime, TriggerFeedback := "PLCMemory".ProductBuffer.MoveFeedback, TriggerMovement => "PLCMemory".ProductBuffer.MoveTrigger, ProductCount => "PLCMemory".ProductBuffer.ProductsCount)
   END_RUNG
   // the same network as SCL:
   IF "Systeem RUN" AND "Tag_31" THEN
       "ProductBuffer_DB"(SensorInput := "Sensor Op Band",   // "ProductBuffer"
                          TimeDelay := "PLCMemory".ProductBuffer.DelayTime,
                          TriggerFeedback := "PLCMemory".ProductBuffer.MoveFeedback,
                          TriggerMovement => "PLCMemory".ProductBuffer.MoveTrigger,
                          ProductCount => "PLCMemory".ProductBuffer.ProductsCount);
   END_IF;
END_REGION

REGION Network 26: ProductBuffer V2
   RUNG wire#powerrail
      Contact( "Systeem RUN" )
      I_Contact( "Tag_31" )
      "ProductBuffer_V2_DB"(SensorInput := "Sensor Op Band", SensorManual := "PositionManagement".Demo_Pos.ManualSensorOverride, TimeDelay := "PLCMemory".ProductBuffer.DelayTime, SystemTime := "PLCMemory".SystemTime, TriggerFeedback := "Move2Done".Q, TriggerMovement => "PLCMemory".ProductBuffer.MoveTrigger, InsertIndex => "PLCMemory".ProductBuffer.InsertIndex, ProductCount => "PLCMemory".ProductBuffer.ProductsCount, SystemTicks =>)
   END_RUNG
   // the same network as SCL:
   IF "Systeem RUN" AND NOT "Tag_31" THEN
       "ProductBuffer_V2_DB"(SensorInput := "Sensor Op Band",   // "ProductBuffer_V2"
                             SensorManual := "PositionManagement".Demo_Pos.ManualSensorOverride,
                             TimeDelay := "PLCMemory".ProductBuffer.DelayTime,
                             SystemTime := "PLCMemory".SystemTime,
                             TriggerFeedback := "Move2Done".Q,
                             TriggerMovement => "PLCMemory".ProductBuffer.MoveTrigger,
                             InsertIndex => "PLCMemory".ProductBuffer.InsertIndex,
                             ProductCount => "PLCMemory".ProductBuffer.ProductsCount);
   END_IF;
END_REGION

REGION Network 27: Speed Select 25%
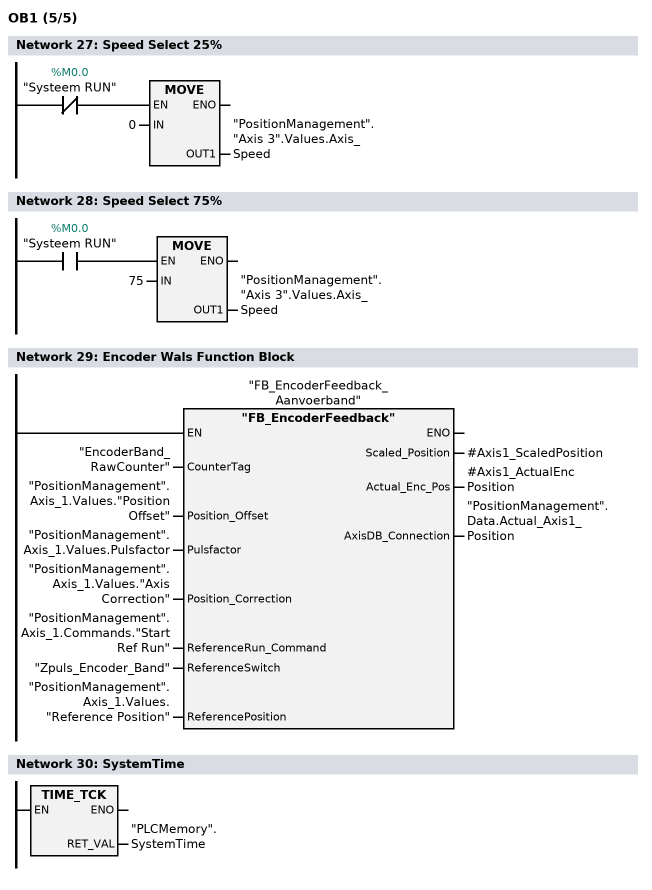
   RUNG wire#powerrail
      I_Contact( "Systeem RUN" )
      { S7_GenerateENO := "TRUE" } Move(in := 0, out1 => "PositionManagement"."Axis 3".Values.Axis_Speed)
   END_RUNG
   // the same network as SCL:
   IF NOT "Systeem RUN" THEN "PositionManagement"."Axis 3".Values.Axis_Speed := 0; END_IF;
END_REGION

REGION Network 28: Speed Select 75%
   RUNG wire#powerrail
      Contact( "Systeem RUN" )
      { S7_GenerateENO := "TRUE" } Move(in := 75, out1 => "PositionManagement"."Axis 3".Values.Axis_Speed)
   END_RUNG
   // the same network as SCL:
   IF "Systeem RUN" THEN "PositionManagement"."Axis 3".Values.Axis_Speed := 75; END_IF;
END_REGION

REGION Network 29: Encoder Wals Function Block
   RUNG wire#powerrail
      "FB_EncoderFeedback_Aanvoerband"(CounterTag := "EncoderBand_RawCounter", Position_Offset := "PositionManagement".Axis_1.Values."Position Offset", Pulsfactor := "PositionManagement".Axis_1.Values.Pulsfactor, Position_Correction := "PositionManagement".Axis_1.Values."Axis Correction", ReferenceRun_Command := "PositionManagement".Axis_1.Commands."Start Ref Run", ReferenceSwitch := "Zpuls_Encoder_Band", ReferencePosition := "PositionManagement".Axis_1.Values."Reference Position", Scaled_Position => #Axis1_ScaledPosition, Actual_Enc_Pos => #Axis1_ActualEncPosition, AxisDB_Connection => "PositionManagement".Data.Actual_Axis1_Position)
   END_RUNG
   // the same network as SCL:
   "FB_EncoderFeedback_Aanvoerband"(CounterTag := "EncoderBand_RawCounter",   // "FB_EncoderFeedback"
                           Position_Offset := "PositionManagement".Axis_1.Values."Position Offset",
                           Pulsfactor := "PositionManagement".Axis_1.Values.Pulsfactor,
                           Position_Correction := "PositionManagement".Axis_1.Values."Axis Correction",
                           ReferenceRun_Command := "PositionManagement".Axis_1.Commands."Start Ref Run",
                           ReferenceSwitch := "Zpuls_Encoder_Band",
                           ReferencePosition := "PositionManagement".Axis_1.Values."Reference Position",
                           Scaled_Position => #Axis1_ScaledPosition,
                           Actual_Enc_Pos => #Axis1_ActualEncPosition,
                           AxisDB_Connection => "PositionManagement".Data.Actual_Axis1_Position);
END_REGION

REGION Network 30: SystemTime
   RUNG wire#powerrail
      TIME_TCK(RET_VAL => "PLCMemory".SystemTime)
   END_RUNG
   // the same network as SCL:
   "PLCMemory".SystemTime := TIME_TCK();
END_REGION
END_ORGANIZATION_BLOCK

FUNCTION "SafetyFunction_Block" : Void   // FC12, LAD
VERSION : 0.1
// stored: AutoNumber true, IsIECCheckEnabled false, UDAEnableTagReadback false
   VAR_INPUT
      "ESB NC Contact" : Bool;
      "ESB NO Contact" : Bool;
      "Reset NO Contact" : Bool;
      "SAFE door 1 NC Contact" : Bool;
      "SAFE door 2 NC Contact" : Bool;
      "Safety Relais NO Contact" : Bool;
   END_VAR
   VAR_OUTPUT
      SAFE_OK_Signal : Bool;
   END_VAR
BEGIN

REGION Network 1: +MC-21K6:1 - Noodstop Circuit
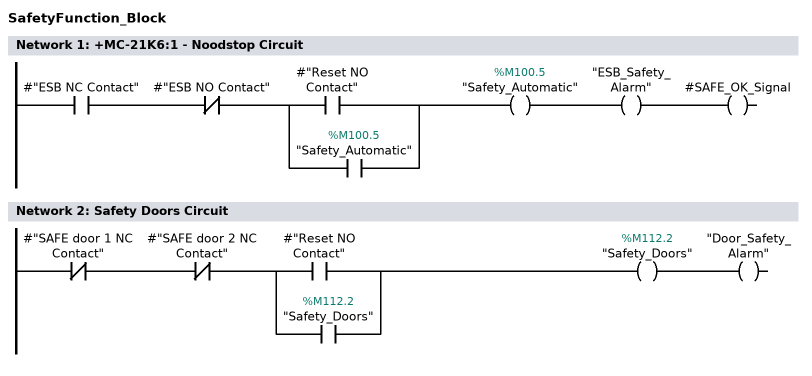
   RUNG wire#powerrail
      Contact( #"ESB NC Contact" )
      I_Contact( #"ESB NO Contact" )
      wire#w1
      Contact( #"Reset NO Contact" )
      wire#w2
      Coil( "Safety_Automatic" )
      Coil( "ESB_Safety_Alarm" )
      Coil( #SAFE_OK_Signal )
   END_RUNG
   RUNG wire#w1
      Contact( "Safety_Automatic" )
   END_RUNG wire#w2
   // the same network as SCL:
   "Safety_Automatic" := #"ESB NC Contact" AND NOT #"ESB NO Contact" AND (#"Reset NO Contact" OR "Safety_Automatic");
   "ESB_Safety_Alarm" := "Safety_Automatic";
   #SAFE_OK_Signal := "Safety_Automatic";
END_REGION

REGION Network 2: Safety Doors Circuit
   RUNG wire#powerrail
      I_Contact( #"SAFE door 1 NC Contact" )
      I_Contact( #"SAFE door 2 NC Contact" )
      wire#w1
      Contact( #"Reset NO Contact" )
      wire#w2
      Coil( "Safety_Doors" )
      Coil( "Door_Safety_Alarm" )
   END_RUNG
   RUNG wire#w1
      Contact( "Safety_Doors" )
   END_RUNG wire#w2
   // the same network as SCL:
   "Safety_Doors" := NOT #"SAFE door 1 NC Contact" AND NOT #"SAFE door 2 NC Contact" AND (#"Reset NO Contact" OR "Safety_Doors");
   "Door_Safety_Alarm" := "Safety_Doors";
END_REGION
END_FUNCTION

FUNCTION "SystemRUN_Block" : Void   // FC13, LAD
VERSION : 0.1
// stored: AutoNumber true, IsIECCheckEnabled false, UDAEnableTagReadback false
   VAR_INPUT
      "Safety Relais Contact" : Bool;
      "Stop Machine NC Contact" : Bool;
      "Fill Magzine Contact" : Bool;
      "Start Machine NO Contact" : Bool;
   END_VAR
   VAR_OUTPUT
      "Run Output Lamp" : Bool;
   END_VAR
BEGIN

REGION Network 1: Systeem RUN
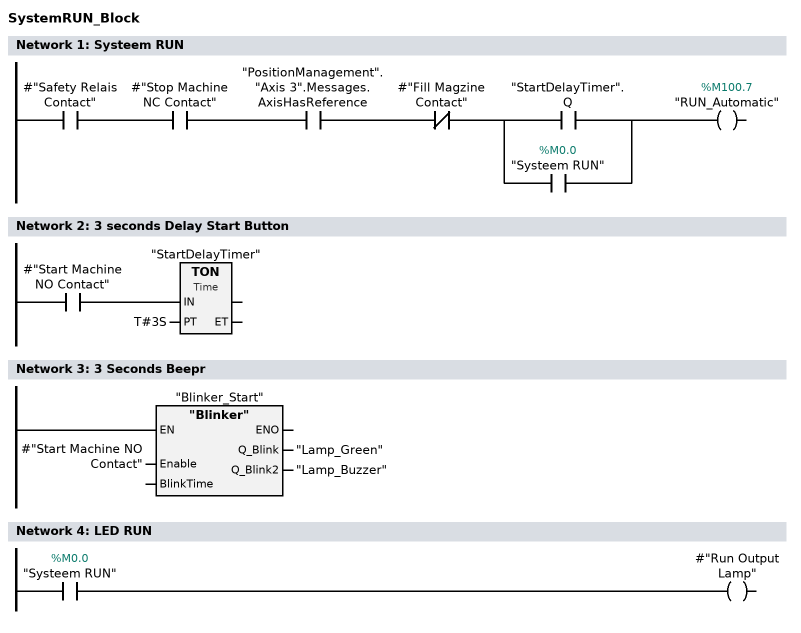
   RUNG wire#powerrail
      Contact( #"Safety Relais Contact" )
      Contact( #"Stop Machine NC Contact" )
      Contact( "PositionManagement"."Axis 3".Messages.AxisHasReference )
      I_Contact( #"Fill Magzine Contact" )
      wire#w1
      Contact( "StartDelayTimer".Q )
      wire#w2
      Coil( "RUN_Automatic" )
   END_RUNG
   RUNG wire#w1
      Contact( "Systeem RUN" )
   END_RUNG wire#w2
   // the same network as SCL:
   "RUN_Automatic" := #"Safety Relais Contact" AND #"Stop Machine NC Contact" AND "PositionManagement"."Axis 3".Messages.AxisHasReference AND NOT #"Fill Magzine Contact" AND ("StartDelayTimer".Q OR "Systeem RUN");
END_REGION

REGION Network 2: 3 seconds Delay Start Button
   RUNG wire#powerrail
      Contact( #"Start Machine NO Contact" )
      { S7_Templates := "time_type := Time" } "StartDelayTimer".TON(pt := T#3S, et =>)
   END_RUNG
   // the same network as SCL:
   "StartDelayTimer".TON(IN := #"Start Machine NO Contact", PT := T#3S);
END_REGION

REGION Network 3: 3 Seconds Beepr
   RUNG wire#powerrail
      "Blinker_Start"(Enable := #"Start Machine NO Contact", BlinkTime :=, Q_Blink => "Lamp_Green", Q_Blink2 => "Lamp_Buzzer")
   END_RUNG
   // the same network as SCL:
   "Blinker_Start"(Enable := #"Start Machine NO Contact", Q_Blink => "Lamp_Green", Q_Blink2 => "Lamp_Buzzer");   // "Blinker"
END_REGION

REGION Network 4: LED RUN
   RUNG wire#powerrail
      Contact( "Systeem RUN" )
      Coil( #"Run Output Lamp" )
   END_RUNG
   // the same network as SCL:
   #"Run Output Lamp" := "Systeem RUN";
END_REGION
END_FUNCTION

FUNCTION "EMStopDrives_Block" : Void   // FC14, LAD
VERSION : 0.1
// stored: AutoNumber true, IsIECCheckEnabled false, UDAEnableTagReadback false
   VAR_INPUT
      "Safety Callback" : Bool;
      Direct_Stop : Bool;
   END_VAR
   VAR_OUTPUT
      "Drive 1 Brake Out" : Bool;
      "Drive 2 Brake Out" : Bool;
      "Drive 3 Brake Out" : Bool;
      "Drive 4 Brake Out" : Bool;
      "Drive 5 Brake Out" : Bool;
      "Drive 6 Brake Out" : Bool;
      "Drive 7 Brake Out" : Bool;
      "Drive 8 Brake Out" : Bool;
      "Drive 9 Brake Out" : Bool;
      "Drive 10 Brake Out" : Bool;
   END_VAR
BEGIN

REGION Network 1: Drives Emergency Stop
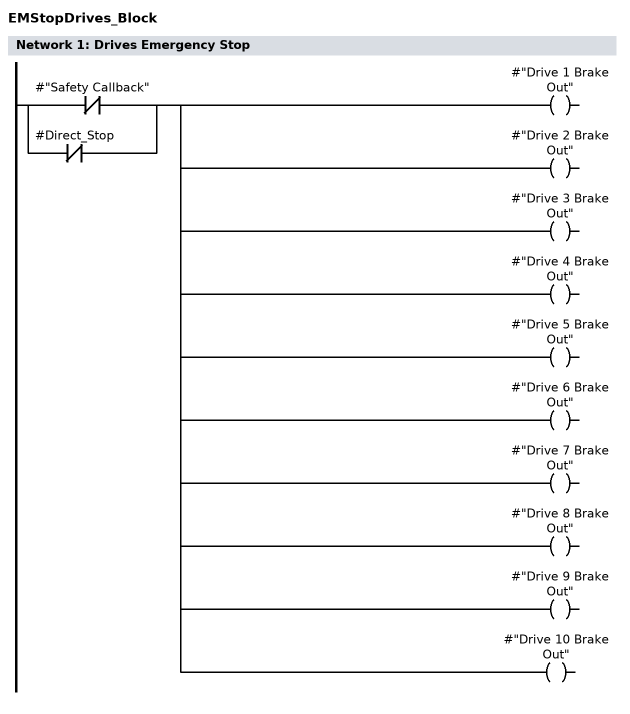
   RUNG wire#powerrail
      I_Contact( #"Safety Callback" )
      wire#w1
      Coil( #"Drive 1 Brake Out" )
   END_RUNG
   RUNG wire#powerrail
      I_Contact( #Direct_Stop )
   END_RUNG wire#w1
   RUNG wire#w1
      Coil( #"Drive 2 Brake Out" )
   END_RUNG
   RUNG wire#w1
      Coil( #"Drive 3 Brake Out" )
   END_RUNG
   RUNG wire#w1
      Coil( #"Drive 4 Brake Out" )
   END_RUNG
   RUNG wire#w1
      Coil( #"Drive 5 Brake Out" )
   END_RUNG
   RUNG wire#w1
      Coil( #"Drive 6 Brake Out" )
   END_RUNG
   RUNG wire#w1
      Coil( #"Drive 7 Brake Out" )
   END_RUNG
   RUNG wire#w1
      Coil( #"Drive 8 Brake Out" )
   END_RUNG
   RUNG wire#w1
      Coil( #"Drive 9 Brake Out" )
   END_RUNG
   RUNG wire#w1
      Coil( #"Drive 10 Brake Out" )
   END_RUNG
   // the same network as SCL:
   #"Drive 1 Brake Out" := NOT #"Safety Callback" OR NOT #Direct_Stop;
   #"Drive 2 Brake Out" := #"Drive 1 Brake Out";
   #"Drive 3 Brake Out" := #"Drive 1 Brake Out";
   #"Drive 4 Brake Out" := #"Drive 1 Brake Out";
   #"Drive 5 Brake Out" := #"Drive 1 Brake Out";
   #"Drive 6 Brake Out" := #"Drive 1 Brake Out";
   #"Drive 7 Brake Out" := #"Drive 1 Brake Out";
   #"Drive 8 Brake Out" := #"Drive 1 Brake Out";
   #"Drive 9 Brake Out" := #"Drive 1 Brake Out";
   #"Drive 10 Brake Out" := #"Drive 1 Brake Out";
END_REGION
END_FUNCTION

FUNCTION "3 - Prog. 1" : Void   // FC1, LAD
TITLE = System Program 1
VERSION : 0.1
// DF
// stored: AutoNumber true, IsIECCheckEnabled false, UDAEnableTagReadback false
   VAR_INPUT
      Axis_3_MovePosition1 : Real;
      Axis_3_MovePosition2 : Real;
   END_VAR
   VAR_OUTPUT
      Axis_On_Pos_1 : Bool;
      Axis_On_Pos_2 : Bool;
   END_VAR
   VAR_TEMP
      TempProdCounter : Int;
      Temp_ProductsToProduce : Bool;
      TimerRunning : Bool;
      ProduceContact : Bool;
      Move2Done : Bool;
      SRWals : Bool;
      Move2Busy : Bool;
      SR_Move2 : Bool;
      Move1Busy : Bool;
      P_TRIG_SnrBand : Bool;
      Temp1 : Bool;
      Min_Pos_1 : Real;
      Max_Pos_1 : Real;
      Min_Pos_2 : Real;
      Max_Pos_2 : Real;
      SR_Move3 : Bool;
      SR_Move1 : Bool;
      AxisToRest : Bool;
      SubDone : Bool;
      P_Trig_ProBehWals : Bool;
      ProductsBehindWals : Int;
      ProductBehindWals : Bool;
      AandrukCilindersOut : Bool;
      Retourband_Delayed : Bool;
      BlowOff_Activated : Bool;
      Pos2_Done : Bool;
      Pos1_Done : Bool;
      ToWaitPosition : Bool;
      BlowOffConf : Bool;
      PTrig_Blow : Bool;
      Move2Done_2 : Bool;
      GoToMove2Pos : Bool;
   END_VAR
   VAR_TEMP   // added for the SCL form of the ladder/FBD networks
      _w1 : Bool;
   END_VAR
BEGIN

REGION Network 1: Set Counter on Zero
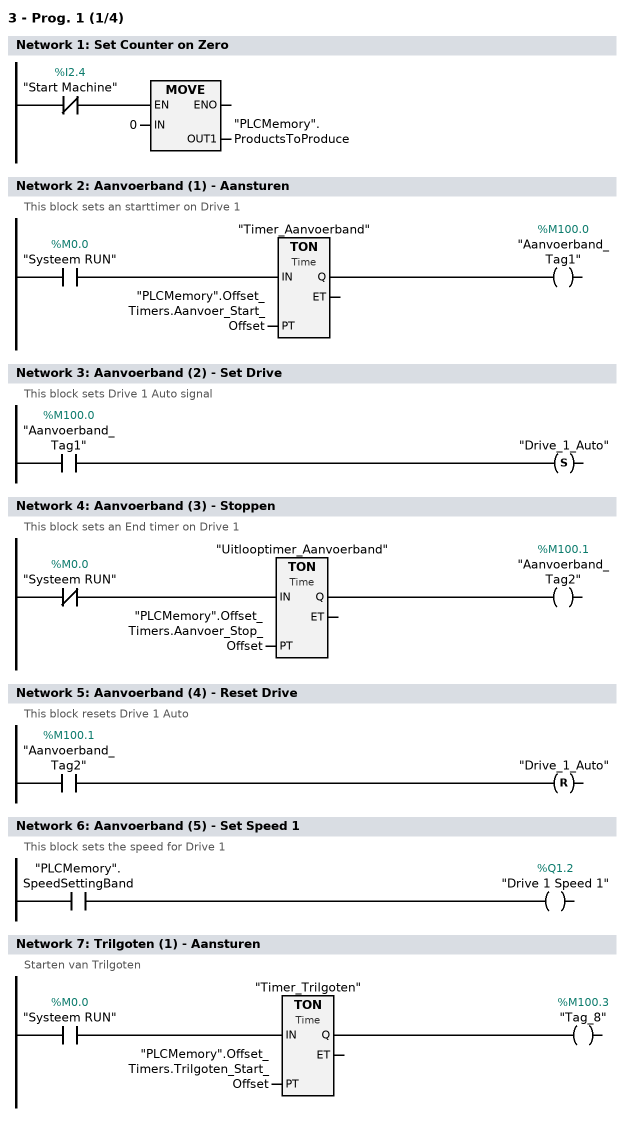
   RUNG wire#powerrail
      I_Contact( "Start Machine" )
      { S7_GenerateENO := "TRUE" } Move(in := 0, out1 => "PLCMemory".ProductsToProduce)
   END_RUNG
   // the same network as SCL:
   IF NOT "Start Machine" THEN "PLCMemory".ProductsToProduce := 0; END_IF;
END_REGION

REGION Network 2: Aanvoerband (1) - Aansturen
   // This block sets an starttimer on Drive 1
   RUNG wire#powerrail
      Contact( "Systeem RUN" )
      { S7_Templates := "time_type := Time" } "Timer_Aanvoerband".TON(pt := "PLCMemory".Offset_Timers.Aanvoer_Start_Offset, et =>)
      Coil( "Aanvoerband_Tag1" )
   END_RUNG
   // the same network as SCL:
   "Timer_Aanvoerband".TON(IN := "Systeem RUN", PT := "PLCMemory".Offset_Timers.Aanvoer_Start_Offset);
   "Aanvoerband_Tag1" := "Timer_Aanvoerband".Q;
END_REGION

REGION Network 3: Aanvoerband (2) - Set Drive
   // This block sets Drive 1 Auto signal
   RUNG wire#powerrail
      Contact( "Aanvoerband_Tag1" )
      S_Coil( "Drive_1_Auto" )
   END_RUNG
   // the same network as SCL:
   IF "Aanvoerband_Tag1" THEN "Drive_1_Auto" := TRUE; END_IF;
END_REGION

REGION Network 4: Aanvoerband (3) - Stoppen
   // This block sets an End timer on Drive 1
   RUNG wire#powerrail
      I_Contact( "Systeem RUN" )
      { S7_Templates := "time_type := Time" } "Uitlooptimer_Aanvoerband".TON(pt := "PLCMemory".Offset_Timers.Aanvoer_Stop_Offset, et =>)
      Coil( "Aanvoerband_Tag2" )
   END_RUNG
   // the same network as SCL:
   "Uitlooptimer_Aanvoerband".TON(IN := NOT "Systeem RUN", PT := "PLCMemory".Offset_Timers.Aanvoer_Stop_Offset);
   "Aanvoerband_Tag2" := "Uitlooptimer_Aanvoerband".Q;
END_REGION

REGION Network 5: Aanvoerband (4) - Reset Drive
   // This block resets Drive 1 Auto
   RUNG wire#powerrail
      Contact( "Aanvoerband_Tag2" )
      R_Coil( "Drive_1_Auto" )
   END_RUNG
   // the same network as SCL:
   IF "Aanvoerband_Tag2" THEN "Drive_1_Auto" := FALSE; END_IF;
END_REGION

REGION Network 6: Aanvoerband (5) - Set Speed 1
   // This block sets the speed for Drive 1
   RUNG wire#powerrail
      Contact( "PLCMemory".SpeedSettingBand )
      Coil( "Drive 1 Speed 1" )
   END_RUNG
   // the same network as SCL:
   "Drive 1 Speed 1" := "PLCMemory".SpeedSettingBand;
END_REGION

REGION Network 7: Trilgoten (1) - Aansturen
   // Starten van Trilgoten
   RUNG wire#powerrail
      Contact( "Systeem RUN" )
      { S7_Templates := "time_type := Time" } "Timer_Trilgoten".TON(pt := "PLCMemory".Offset_Timers.Trilgoten_Start_Offset, et =>)
      Coil( "Tag_8" )
   END_RUNG
   // the same network as SCL:
   "Timer_Trilgoten".TON(IN := "Systeem RUN", PT := "PLCMemory".Offset_Timers.Trilgoten_Start_Offset);
   "Tag_8" := "Timer_Trilgoten".Q;
END_REGION

REGION Network 8: Trilgoten (2) - Set Drive
   // Set drive Trilgoten (Drive 2)
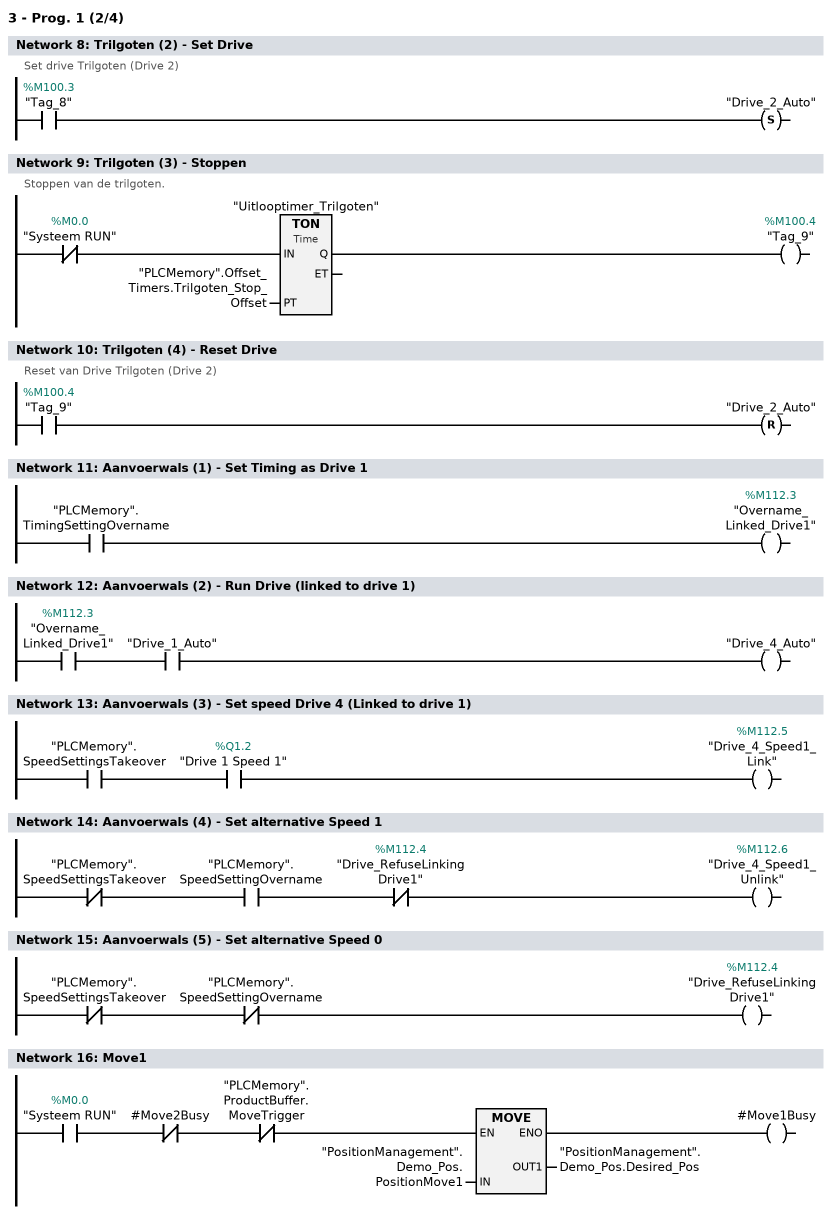
   RUNG wire#powerrail
      Contact( "Tag_8" )
      S_Coil( "Drive_2_Auto" )
   END_RUNG
   // the same network as SCL:
   IF "Tag_8" THEN "Drive_2_Auto" := TRUE; END_IF;
END_REGION

REGION Network 9: Trilgoten (3) - Stoppen
   // Stoppen van de trilgoten.
   RUNG wire#powerrail
      I_Contact( "Systeem RUN" )
      { S7_Templates := "time_type := Time" } "Uitlooptimer_Trilgoten".TON(pt := "PLCMemory".Offset_Timers.Trilgoten_Stop_Offset, et =>)
      Coil( "Tag_9" )
   END_RUNG
   // the same network as SCL:
   "Uitlooptimer_Trilgoten".TON(IN := NOT "Systeem RUN", PT := "PLCMemory".Offset_Timers.Trilgoten_Stop_Offset);
   "Tag_9" := "Uitlooptimer_Trilgoten".Q;
END_REGION

REGION Network 10: Trilgoten (4) - Reset Drive
   // Reset van Drive Trilgoten (Drive 2)
   RUNG wire#powerrail
      Contact( "Tag_9" )
      R_Coil( "Drive_2_Auto" )
   END_RUNG
   // the same network as SCL:
   IF "Tag_9" THEN "Drive_2_Auto" := FALSE; END_IF;
END_REGION

REGION Network 11: Aanvoerwals (1) - Set Timing as Drive 1
   RUNG wire#powerrail
      Contact( "PLCMemory".TimingSettingOvername )
      Coil( "Overname_Linked_Drive1" )
   END_RUNG
   // the same network as SCL:
   "Overname_Linked_Drive1" := "PLCMemory".TimingSettingOvername;
END_REGION

REGION Network 12: Aanvoerwals (2) - Run Drive (linked to drive 1)
   RUNG wire#powerrail
      Contact( "Overname_Linked_Drive1" )
      Contact( "Drive_1_Auto" )
      Coil( "Drive_4_Auto" )
   END_RUNG
   // the same network as SCL:
   "Drive_4_Auto" := "Overname_Linked_Drive1" AND "Drive_1_Auto";
END_REGION

REGION Network 13: Aanvoerwals (3) - Set speed Drive 4 (Linked to drive 1)
   RUNG wire#powerrail
      Contact( "PLCMemory".SpeedSettingsTakeover )
      Contact( "Drive 1 Speed 1" )
      Coil( "Drive_4_Speed1_Link" )
   END_RUNG
   // the same network as SCL:
   "Drive_4_Speed1_Link" := "PLCMemory".SpeedSettingsTakeover AND "Drive 1 Speed 1";
END_REGION

REGION Network 14: Aanvoerwals (4) - Set alternative Speed 1
   RUNG wire#powerrail
      I_Contact( "PLCMemory".SpeedSettingsTakeover )
      Contact( "PLCMemory".SpeedSettingOvername )
      I_Contact( "Drive_RefuseLinkingDrive1" )
      Coil( "Drive_4_Speed1_Unlink" )
   END_RUNG
   // the same network as SCL:
   "Drive_4_Speed1_Unlink" := NOT "PLCMemory".SpeedSettingsTakeover AND "PLCMemory".SpeedSettingOvername AND NOT "Drive_RefuseLinkingDrive1";
END_REGION

REGION Network 15: Aanvoerwals (5) - Set alternative Speed 0
   RUNG wire#powerrail
      I_Contact( "PLCMemory".SpeedSettingsTakeover )
      I_Contact( "PLCMemory".SpeedSettingOvername )
      Coil( "Drive_RefuseLinkingDrive1" )
   END_RUNG
   // the same network as SCL:
   "Drive_RefuseLinkingDrive1" := NOT "PLCMemory".SpeedSettingsTakeover AND NOT "PLCMemory".SpeedSettingOvername;
END_REGION

REGION Network 16: Move1
   RUNG wire#powerrail
      Contact( "Systeem RUN" )
      I_Contact( #Move2Busy )
      I_Contact( "PLCMemory".ProductBuffer.MoveTrigger )
      { S7_GenerateENO := "TRUE" } Move(in := "PositionManagement".Demo_Pos.PositionMove1, out1 => "PositionManagement".Demo_Pos.Desired_Pos)
      Coil( #Move1Busy )
   END_RUNG
   // the same network as SCL:
   // ENO of a box is taken as its EN; it also drops when the box reports an error
   #_w1 := "Systeem RUN" AND NOT #Move2Busy AND NOT "PLCMemory".ProductBuffer.MoveTrigger;
   IF #_w1 THEN
       "PositionManagement".Demo_Pos.Desired_Pos := "PositionManagement".Demo_Pos.PositionMove1;
   END_IF;
   #Move1Busy := #_w1;
END_REGION

REGION Network 17: Move 2
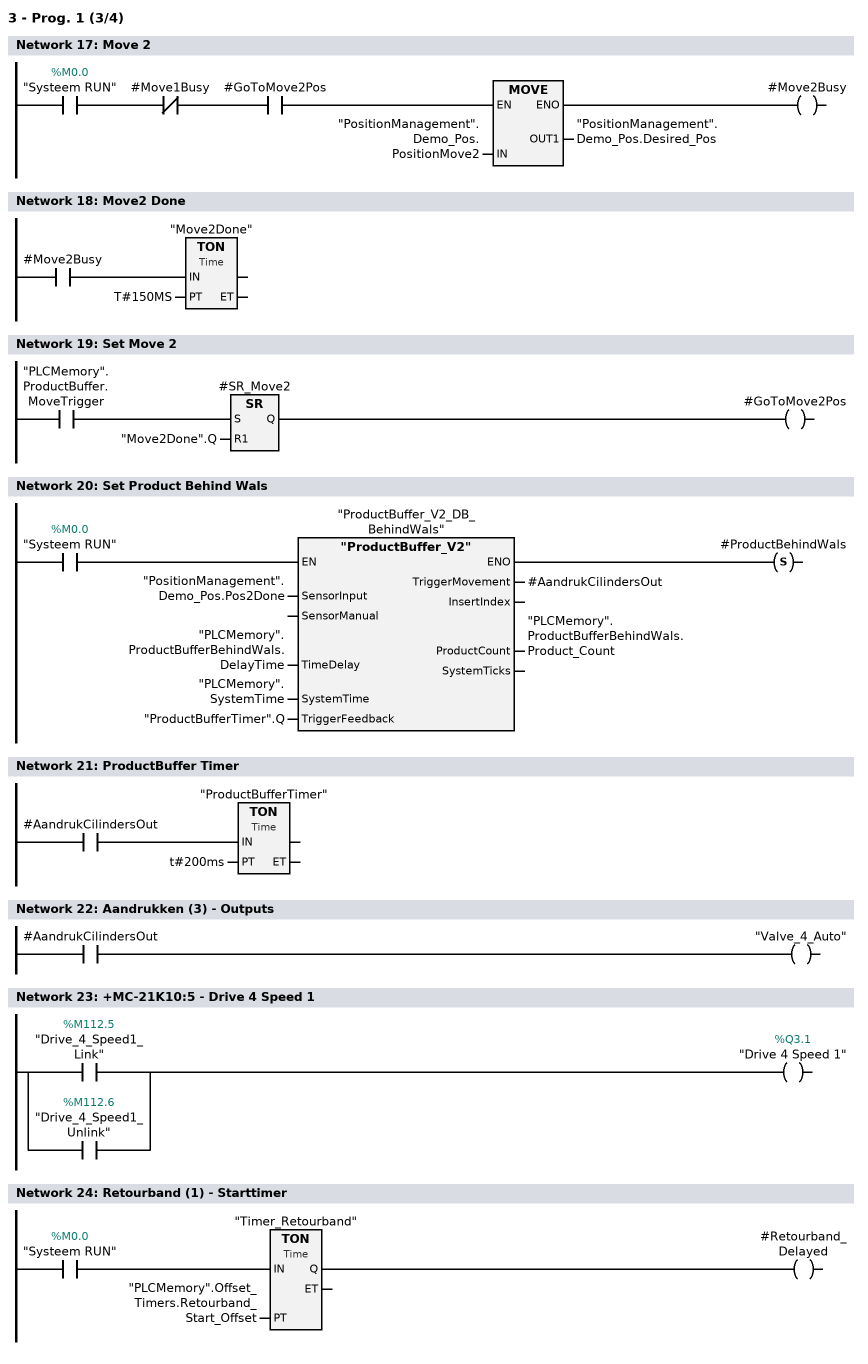
   RUNG wire#powerrail
      Contact( "Systeem RUN" )
      I_Contact( #Move1Busy )
      Contact( #GoToMove2Pos )
      { S7_GenerateENO := "TRUE" } Move(in := "PositionManagement".Demo_Pos.PositionMove2, out1 => "PositionManagement".Demo_Pos.Desired_Pos)
      Coil( #Move2Busy )
   END_RUNG
   // the same network as SCL:
   // ENO of a box is taken as its EN; it also drops when the box reports an error
   #_w1 := "Systeem RUN" AND NOT #Move1Busy AND #GoToMove2Pos;
   IF #_w1 THEN
       "PositionManagement".Demo_Pos.Desired_Pos := "PositionManagement".Demo_Pos.PositionMove2;
   END_IF;
   #Move2Busy := #_w1;
END_REGION

REGION Network 18: Move2 Done
   RUNG wire#powerrail
      Contact( #Move2Busy )
      { S7_Templates := "time_type := Time" } "Move2Done".TON(pt := T#150MS, et =>)
   END_RUNG
   // the same network as SCL:
   "Move2Done".TON(IN := #Move2Busy, PT := T#150MS);
END_REGION

REGION Network 19: Set Move 2
   RUNG wire#powerrail
      Contact( "PLCMemory".ProductBuffer.MoveTrigger )
      S_SR(operand := #SR_Move2, r1 := "Move2Done".Q)
      Coil( #GoToMove2Pos )
   END_RUNG
   // the same network as SCL:
   IF "PLCMemory".ProductBuffer.MoveTrigger THEN
       #SR_Move2 := TRUE;   // SR flip-flop
   END_IF;
   IF "Move2Done".Q THEN #SR_Move2 := FALSE; END_IF;
   #GoToMove2Pos := #SR_Move2;
END_REGION

REGION Network 20: Set Product Behind Wals
   RUNG wire#powerrail
      Contact( "Systeem RUN" )
      "ProductBuffer_V2_DB_BehindWals"(SensorInput := "PositionManagement".Demo_Pos.Pos2Done, SensorManual :=, TimeDelay := "PLCMemory".ProductBufferBehindWals.DelayTime, SystemTime := "PLCMemory".SystemTime, TriggerFeedback := "ProductBufferTimer".Q, TriggerMovement => #AandrukCilindersOut, InsertIndex =>, ProductCount => "PLCMemory".ProductBufferBehindWals.Product_Count, SystemTicks =>)
      S_Coil( #ProductBehindWals )
   END_RUNG
   // the same network as SCL:
   "ProductBuffer_V2_DB_BehindWals"(EN := "Systeem RUN",   // "ProductBuffer_V2"
                           SensorInput := "PositionManagement".Demo_Pos.Pos2Done,
                           TimeDelay := "PLCMemory".ProductBufferBehindWals.DelayTime,
                           SystemTime := "PLCMemory".SystemTime,
                           TriggerFeedback := "ProductBufferTimer".Q,
                           TriggerMovement => #AandrukCilindersOut,
                           ProductCount => "PLCMemory".ProductBufferBehindWals.Product_Count,
                           ENO => #_w1);
   IF #_w1 THEN #ProductBehindWals := TRUE; END_IF;
END_REGION

REGION Network 21: ProductBuffer Timer
   RUNG wire#powerrail
      Contact( #AandrukCilindersOut )
      { S7_Templates := "time_type := Time" } "ProductBufferTimer".TON(pt := t#200ms, et =>)
   END_RUNG
   // the same network as SCL:
   "ProductBufferTimer".TON(IN := #AandrukCilindersOut, PT := t#200ms);
END_REGION

REGION Network 22: Aandrukken (3) - Outputs
   RUNG wire#powerrail
      Contact( #AandrukCilindersOut )
      Coil( "Valve_4_Auto" )
   END_RUNG
   // the same network as SCL:
   "Valve_4_Auto" := #AandrukCilindersOut;
END_REGION

REGION Network 23: +MC-21K10:5 - Drive 4 Speed 1
   RUNG wire#powerrail
      Contact( "Drive_4_Speed1_Link" )
      wire#w1
      Coil( "Drive 4 Speed 1" )
   END_RUNG
   RUNG wire#powerrail
      Contact( "Drive_4_Speed1_Unlink" )
   END_RUNG wire#w1
   // the same network as SCL:
   "Drive 4 Speed 1" := "Drive_4_Speed1_Link" OR "Drive_4_Speed1_Unlink";
END_REGION

REGION Network 24: Retourband (1) - Starttimer
   RUNG wire#powerrail
      Contact( "Systeem RUN" )
      { S7_Templates := "time_type := Time" } "Timer_Retourband".TON(pt := "PLCMemory".Offset_Timers.Retourband_Start_Offset, et =>)
      Coil( #Retourband_Delayed )
   END_RUNG
   // the same network as SCL:
   "Timer_Retourband".TON(IN := "Systeem RUN", PT := "PLCMemory".Offset_Timers.Retourband_Start_Offset);
   #Retourband_Delayed := "Timer_Retourband".Q;
END_REGION

REGION Network 25: Retourband (2) - Start Drive
   // This block sets Drive 1 Auto signal
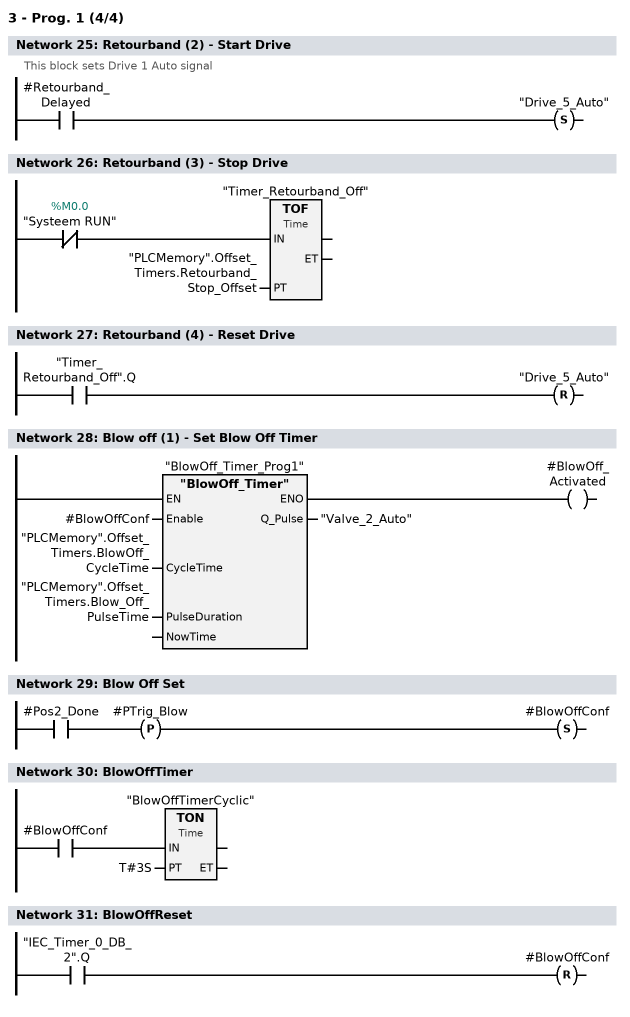
   RUNG wire#powerrail
      Contact( #Retourband_Delayed )
      S_Coil( "Drive_5_Auto" )
   END_RUNG
   // the same network as SCL:
   IF #Retourband_Delayed THEN "Drive_5_Auto" := TRUE; END_IF;
END_REGION

REGION Network 26: Retourband (3) - Stop Drive
   RUNG wire#powerrail
      I_Contact( "Systeem RUN" )
      { S7_Templates := "time_type := Time" } "Timer_Retourband_Off".TOF(pt := "PLCMemory".Offset_Timers.Retourband_Stop_Offset, et =>)
   END_RUNG
   // the same network as SCL:
   "Timer_Retourband_Off".TOF(IN := NOT "Systeem RUN", PT := "PLCMemory".Offset_Timers.Retourband_Stop_Offset);
END_REGION

REGION Network 27: Retourband (4) - Reset Drive
   RUNG wire#powerrail
      Contact( "Timer_Retourband_Off".Q )
      R_Coil( "Drive_5_Auto" )
   END_RUNG
   // the same network as SCL:
   IF "Timer_Retourband_Off".Q THEN "Drive_5_Auto" := FALSE; END_IF;
END_REGION

REGION Network 28: Blow off (1) - Set Blow Off Timer
   RUNG wire#powerrail
      "BlowOff_Timer_Prog1"(Enable := #BlowOffConf, CycleTime := "PLCMemory".Offset_Timers.BlowOff_CycleTime, PulseDuration := "PLCMemory".Offset_Timers.Blow_Off_PulseTime, NowTime :=, Q_Pulse => "Valve_2_Auto")
      Coil( #BlowOff_Activated )
   END_RUNG
   // the same network as SCL:
   "BlowOff_Timer_Prog1"(Enable := #BlowOffConf,   // "BlowOff_Timer"
                         CycleTime := "PLCMemory".Offset_Timers.BlowOff_CycleTime,
                         PulseDuration := "PLCMemory".Offset_Timers.Blow_Off_PulseTime,
                         Q_Pulse => "Valve_2_Auto",
                         ENO => #_w1);
   #BlowOff_Activated := #_w1;
END_REGION

REGION Network 29: Blow Off Set
   RUNG wire#powerrail
      Contact( #Pos2_Done )
      P_Trig( #PTrig_Blow )
      S_Coil( #BlowOffConf )
   END_RUNG
   // the same network as SCL:
   #_w1 := #Pos2_Done AND NOT #PTrig_Blow;   // rising edge
   #PTrig_Blow := #Pos2_Done;
   IF #_w1 THEN #BlowOffConf := TRUE; END_IF;
END_REGION

REGION Network 30: BlowOffTimer
   RUNG wire#powerrail
      Contact( #BlowOffConf )
      { S7_Templates := "time_type := Time" } "BlowOffTimerCyclic".TON(pt := T#3S, et =>)
   END_RUNG
   // the same network as SCL:
   "BlowOffTimerCyclic".TON(IN := #BlowOffConf, PT := T#3S);
END_REGION

REGION Network 31: BlowOffReset
   RUNG wire#powerrail
      Contact( "IEC_Timer_0_DB_2".Q )
      R_Coil( #BlowOffConf )
   END_RUNG
   // the same network as SCL:
   IF "IEC_Timer_0_DB_2".Q THEN #BlowOffConf := FALSE; END_IF;
END_REGION
END_FUNCTION

FUNCTION "4 - Prog. 2" : Void   // FC2, LAD
TITLE = System Program 2
VERSION : 0.1
// stored: AutoNumber true, IsIECCheckEnabled false, UDAEnableTagReadback false
BEGIN

REGION Network 1: Close 1 Magazine Hole (cilinder)
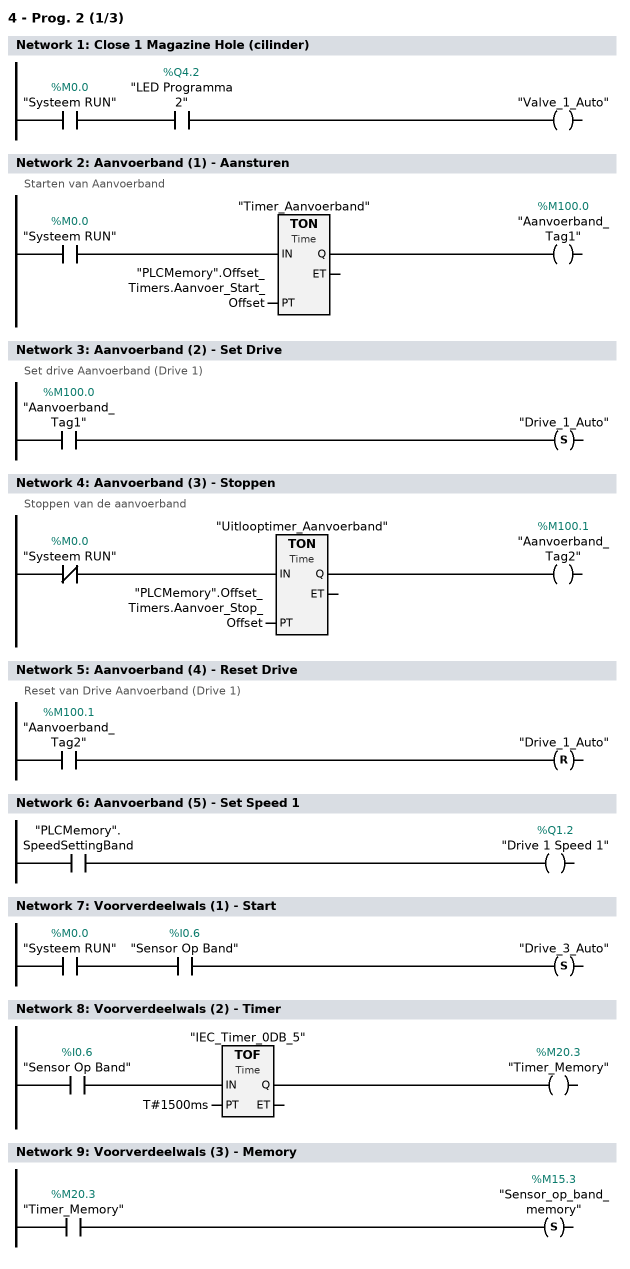
   RUNG wire#powerrail
      Contact( "Systeem RUN" )
      Contact( "LED Programma 2" )
      Coil( "Valve_1_Auto" )
   END_RUNG
   // the same network as SCL:
   "Valve_1_Auto" := "Systeem RUN" AND "LED Programma 2";
END_REGION

REGION Network 2: Aanvoerband (1) - Aansturen
   // Starten van Aanvoerband
   RUNG wire#powerrail
      Contact( "Systeem RUN" )
      { S7_Templates := "time_type := Time" } "Timer_Aanvoerband".TON(pt := "PLCMemory".Offset_Timers.Aanvoer_Start_Offset, et =>)
      Coil( "Aanvoerband_Tag1" )
   END_RUNG
   // the same network as SCL:
   "Timer_Aanvoerband".TON(IN := "Systeem RUN", PT := "PLCMemory".Offset_Timers.Aanvoer_Start_Offset);
   "Aanvoerband_Tag1" := "Timer_Aanvoerband".Q;
END_REGION

REGION Network 3: Aanvoerband (2) - Set Drive
   // Set drive Aanvoerband (Drive 1)
   RUNG wire#powerrail
      Contact( "Aanvoerband_Tag1" )
      S_Coil( "Drive_1_Auto" )
   END_RUNG
   // the same network as SCL:
   IF "Aanvoerband_Tag1" THEN "Drive_1_Auto" := TRUE; END_IF;
END_REGION

REGION Network 4: Aanvoerband (3) - Stoppen
   // Stoppen van de aanvoerband
   RUNG wire#powerrail
      I_Contact( "Systeem RUN" )
      { S7_Templates := "time_type := Time" } "Uitlooptimer_Aanvoerband".TON(pt := "PLCMemory".Offset_Timers.Aanvoer_Stop_Offset, et =>)
      Coil( "Aanvoerband_Tag2" )
   END_RUNG
   // the same network as SCL:
   "Uitlooptimer_Aanvoerband".TON(IN := NOT "Systeem RUN", PT := "PLCMemory".Offset_Timers.Aanvoer_Stop_Offset);
   "Aanvoerband_Tag2" := "Uitlooptimer_Aanvoerband".Q;
END_REGION

REGION Network 5: Aanvoerband (4) - Reset Drive
   // Reset van Drive Aanvoerband (Drive 1)
   RUNG wire#powerrail
      Contact( "Aanvoerband_Tag2" )
      R_Coil( "Drive_1_Auto" )
   END_RUNG
   // the same network as SCL:
   IF "Aanvoerband_Tag2" THEN "Drive_1_Auto" := FALSE; END_IF;
END_REGION

REGION Network 6: Aanvoerband (5) - Set Speed 1
   RUNG wire#powerrail
      Contact( "PLCMemory".SpeedSettingBand )
      Coil( "Drive 1 Speed 1" )
   END_RUNG
   // the same network as SCL:
   "Drive 1 Speed 1" := "PLCMemory".SpeedSettingBand;
END_REGION

REGION Network 7: Voorverdeelwals (1) - Start
   RUNG wire#powerrail
      Contact( "Systeem RUN" )
      Contact( "Sensor Op Band" )
      S_Coil( "Drive_3_Auto" )
   END_RUNG
   // the same network as SCL:
   IF "Systeem RUN" AND "Sensor Op Band" THEN "Drive_3_Auto" := TRUE; END_IF;
END_REGION

REGION Network 8: Voorverdeelwals (2) - Timer
   RUNG wire#powerrail
      Contact( "Sensor Op Band" )
      { S7_Templates := "time_type := Time" } "IEC_Timer_0DB_5".TOF(pt := T#1500ms, et =>)
      Coil( "Timer_Memory" )
   END_RUNG
   // the same network as SCL:
   "IEC_Timer_0DB_5".TOF(IN := "Sensor Op Band", PT := T#1500ms);
   "Timer_Memory" := "IEC_Timer_0DB_5".Q;
END_REGION

REGION Network 9: Voorverdeelwals (3) - Memory
   RUNG wire#powerrail
      Contact( "Timer_Memory" )
      S_Coil( "Sensor_op_band_memory" )
   END_RUNG
   // the same network as SCL:
   IF "Timer_Memory" THEN "Sensor_op_band_memory" := TRUE; END_IF;
END_REGION

REGION Network 10: Voorverdeelwals (4) - Delaying
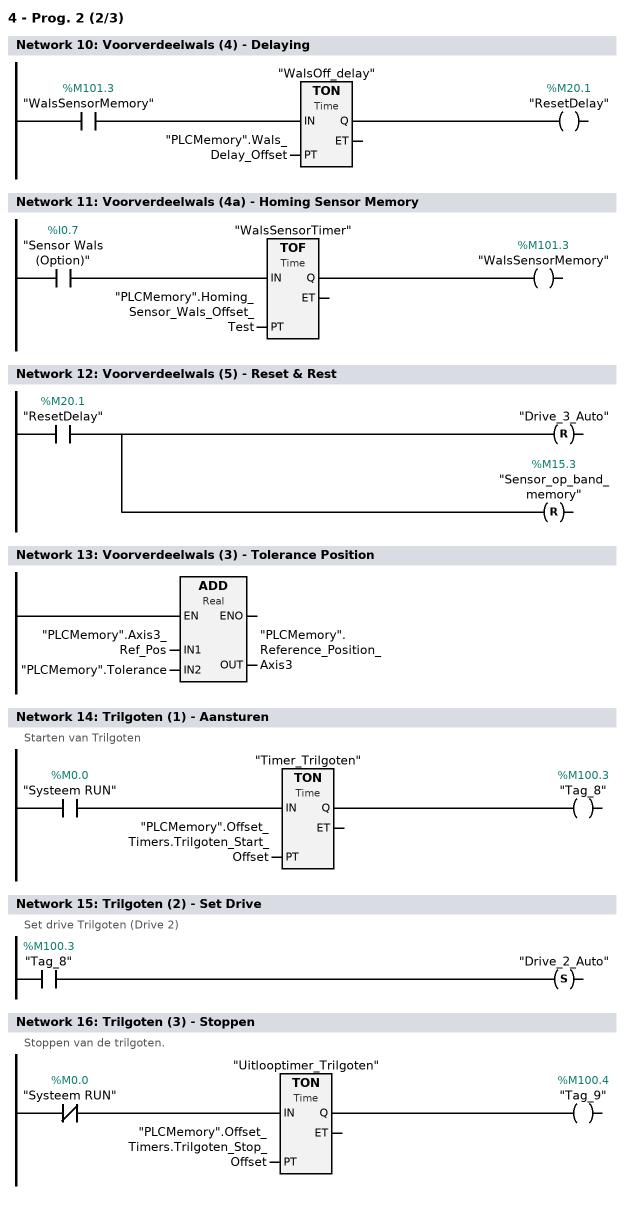
   RUNG wire#powerrail
      Contact( "WalsSensorMemory" )
      { S7_Templates := "time_type := Time" } "WalsOff_delay".TON(pt := "PLCMemory".Wals_Delay_Offset, et =>)
      Coil( "ResetDelay" )
   END_RUNG
   // the same network as SCL:
   "WalsOff_delay".TON(IN := "WalsSensorMemory", PT := "PLCMemory".Wals_Delay_Offset);
   "ResetDelay" := "WalsOff_delay".Q;
END_REGION

REGION Network 11: Voorverdeelwals (4a) - Homing Sensor Memory
   RUNG wire#powerrail
      Contact( "Sensor Wals (Option)" )
      { S7_Templates := "time_type := Time" } "WalsSensorTimer".TOF(pt := "PLCMemory".Homing_Sensor_Wals_Offset_Test, et =>)
      Coil( "WalsSensorMemory" )
   END_RUNG
   // the same network as SCL:
   "WalsSensorTimer".TOF(IN := "Sensor Wals (Option)", PT := "PLCMemory".Homing_Sensor_Wals_Offset_Test);
   "WalsSensorMemory" := "WalsSensorTimer".Q;
END_REGION

REGION Network 12: Voorverdeelwals (5) - Reset & Rest
   RUNG wire#powerrail
      Contact( "ResetDelay" )
      wire#w1
      R_Coil( "Drive_3_Auto" )
   END_RUNG
   RUNG wire#w1
      R_Coil( "Sensor_op_band_memory" )
   END_RUNG
   // the same network as SCL:
   IF "ResetDelay" THEN
       "Drive_3_Auto" := FALSE;
       "Sensor_op_band_memory" := FALSE;
   END_IF;
END_REGION

REGION Network 13: Voorverdeelwals (3) - Tolerance Position
   RUNG wire#powerrail
      { S7_Templates := "SrcType := Real"; S7_GenerateENO := "TRUE" } Add(in1 := "PLCMemory".Axis3_Ref_Pos, in2 := "PLCMemory".Tolerance, out => "PLCMemory".Reference_Position_Axis3)
   END_RUNG
   // the same network as SCL:
   "PLCMemory".Reference_Position_Axis3 := "PLCMemory".Axis3_Ref_Pos + "PLCMemory".Tolerance;
END_REGION

REGION Network 14: Trilgoten (1) - Aansturen
   // Starten van Trilgoten
   RUNG wire#powerrail
      Contact( "Systeem RUN" )
      { S7_Templates := "time_type := Time" } "Timer_Trilgoten".TON(pt := "PLCMemory".Offset_Timers.Trilgoten_Start_Offset, et =>)
      Coil( "Tag_8" )
   END_RUNG
   // the same network as SCL:
   "Timer_Trilgoten".TON(IN := "Systeem RUN", PT := "PLCMemory".Offset_Timers.Trilgoten_Start_Offset);
   "Tag_8" := "Timer_Trilgoten".Q;
END_REGION

REGION Network 15: Trilgoten (2) - Set Drive
   // Set drive Trilgoten (Drive 2)
   RUNG wire#powerrail
      Contact( "Tag_8" )
      S_Coil( "Drive_2_Auto" )
   END_RUNG
   // the same network as SCL:
   IF "Tag_8" THEN "Drive_2_Auto" := TRUE; END_IF;
END_REGION

REGION Network 16: Trilgoten (3) - Stoppen
   // Stoppen van de trilgoten.
   RUNG wire#powerrail
      I_Contact( "Systeem RUN" )
      { S7_Templates := "time_type := Time" } "Uitlooptimer_Trilgoten".TON(pt := "PLCMemory".Offset_Timers.Trilgoten_Stop_Offset, et =>)
      Coil( "Tag_9" )
   END_RUNG
   // the same network as SCL:
   "Uitlooptimer_Trilgoten".TON(IN := NOT "Systeem RUN", PT := "PLCMemory".Offset_Timers.Trilgoten_Stop_Offset);
   "Tag_9" := "Uitlooptimer_Trilgoten".Q;
END_REGION

REGION Network 17: Trilgoten (4) - Reset Drive
   // Reset van Drive Trilgoten (Drive 2)
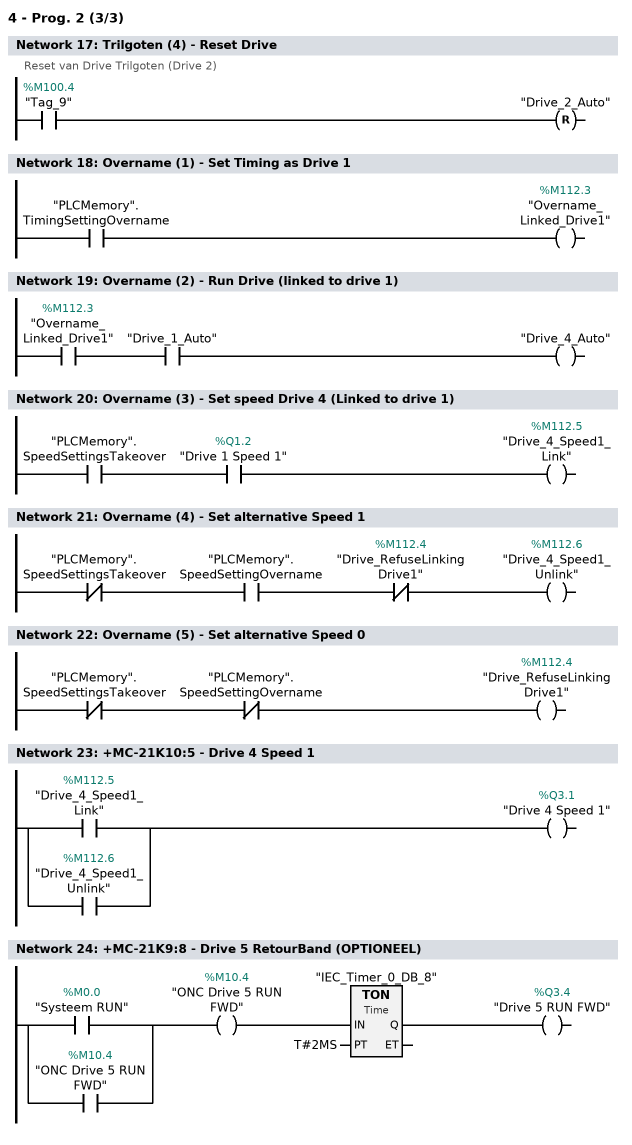
   RUNG wire#powerrail
      Contact( "Tag_9" )
      R_Coil( "Drive_2_Auto" )
   END_RUNG
   // the same network as SCL:
   IF "Tag_9" THEN "Drive_2_Auto" := FALSE; END_IF;
END_REGION

REGION Network 18: Overname (1) - Set Timing as Drive 1
   RUNG wire#powerrail
      Contact( "PLCMemory".TimingSettingOvername )
      Coil( "Overname_Linked_Drive1" )
   END_RUNG
   // the same network as SCL:
   "Overname_Linked_Drive1" := "PLCMemory".TimingSettingOvername;
END_REGION

REGION Network 19: Overname (2) - Run Drive (linked to drive 1)
   RUNG wire#powerrail
      Contact( "Overname_Linked_Drive1" )
      Contact( "Drive_1_Auto" )
      Coil( "Drive_4_Auto" )
   END_RUNG
   // the same network as SCL:
   "Drive_4_Auto" := "Overname_Linked_Drive1" AND "Drive_1_Auto";
END_REGION

REGION Network 20: Overname (3) - Set speed Drive 4 (Linked to drive 1)
   RUNG wire#powerrail
      Contact( "PLCMemory".SpeedSettingsTakeover )
      Contact( "Drive 1 Speed 1" )
      Coil( "Drive_4_Speed1_Link" )
   END_RUNG
   // the same network as SCL:
   "Drive_4_Speed1_Link" := "PLCMemory".SpeedSettingsTakeover AND "Drive 1 Speed 1";
END_REGION

REGION Network 21: Overname (4) - Set alternative Speed 1
   RUNG wire#powerrail
      I_Contact( "PLCMemory".SpeedSettingsTakeover )
      Contact( "PLCMemory".SpeedSettingOvername )
      I_Contact( "Drive_RefuseLinkingDrive1" )
      Coil( "Drive_4_Speed1_Unlink" )
   END_RUNG
   // the same network as SCL:
   "Drive_4_Speed1_Unlink" := NOT "PLCMemory".SpeedSettingsTakeover AND "PLCMemory".SpeedSettingOvername AND NOT "Drive_RefuseLinkingDrive1";
END_REGION

REGION Network 22: Overname (5) - Set alternative Speed 0
   RUNG wire#powerrail
      I_Contact( "PLCMemory".SpeedSettingsTakeover )
      I_Contact( "PLCMemory".SpeedSettingOvername )
      Coil( "Drive_RefuseLinkingDrive1" )
   END_RUNG
   // the same network as SCL:
   "Drive_RefuseLinkingDrive1" := NOT "PLCMemory".SpeedSettingsTakeover AND NOT "PLCMemory".SpeedSettingOvername;
END_REGION

REGION Network 23: +MC-21K10:5 - Drive 4 Speed 1
   RUNG wire#powerrail
      Contact( "Drive_4_Speed1_Link" )
      wire#w1
      Coil( "Drive 4 Speed 1" )
   END_RUNG
   RUNG wire#powerrail
      Contact( "Drive_4_Speed1_Unlink" )
   END_RUNG wire#w1
   // the same network as SCL:
   "Drive 4 Speed 1" := "Drive_4_Speed1_Link" OR "Drive_4_Speed1_Unlink";
END_REGION

REGION Network 24: +MC-21K9:8 - Drive 5 RetourBand (OPTIONEEL)
   RUNG wire#powerrail
      Contact( "Systeem RUN" )
      wire#w1
      Coil( "ONC Drive 5 RUN FWD" )
      { S7_Templates := "time_type := Time" } "IEC_Timer_0_DB_8".TON(pt := T#2MS, et =>)
      Coil( "Drive 5 RUN FWD" )
   END_RUNG
   RUNG wire#powerrail
      Contact( "ONC Drive 5 RUN FWD" )
   END_RUNG wire#w1
   // the same network as SCL:
   "ONC Drive 5 RUN FWD" := "Systeem RUN" OR "ONC Drive 5 RUN FWD";
   "IEC_Timer_0_DB_8".TON(IN := "ONC Drive 5 RUN FWD", PT := T#2MS);
   "Drive 5 RUN FWD" := "IEC_Timer_0_DB_8".Q;
END_REGION
END_FUNCTION

FUNCTION "5 - Prog. 3" : Void   // FC3, LAD
TITLE = System Program 3
VERSION : 0.1
// stored: AutoNumber true, IsIECCheckEnabled false, UDAEnableTagReadback false
BEGIN

REGION Network 1: Close 1 Magazine Hole (cilinder)
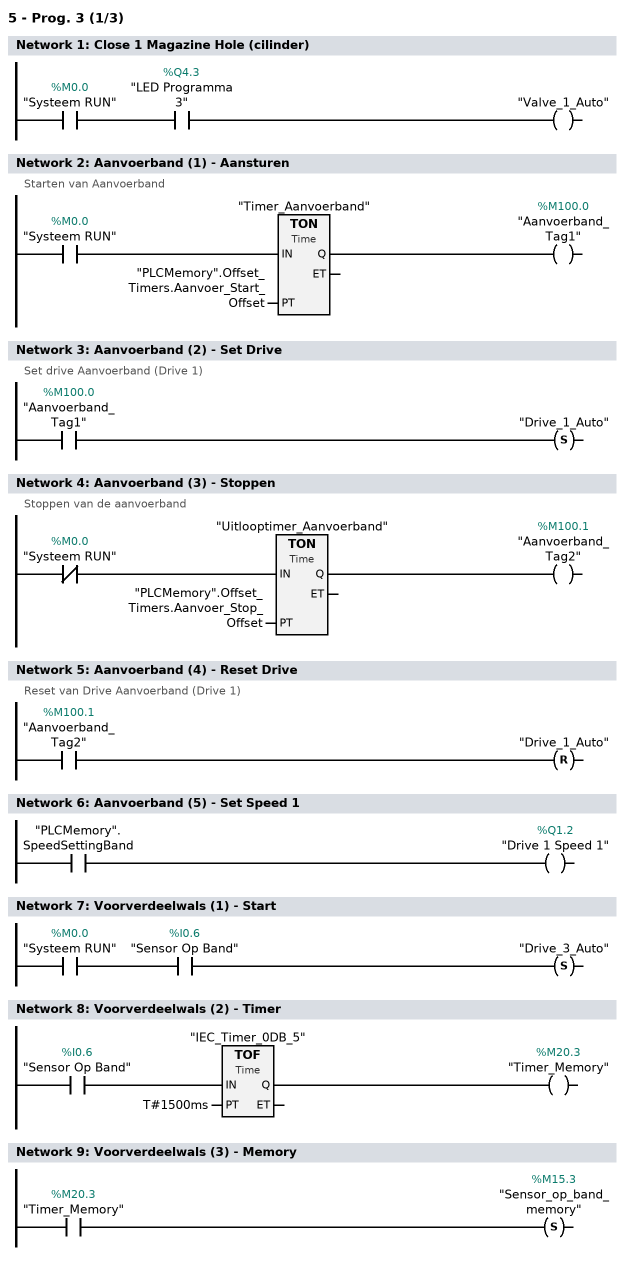
   RUNG wire#powerrail
      Contact( "Systeem RUN" )
      Contact( "LED Programma 3" )
      Coil( "Valve_1_Auto" )
   END_RUNG
   // the same network as SCL:
   "Valve_1_Auto" := "Systeem RUN" AND "LED Programma 3";
END_REGION

REGION Network 2: Aanvoerband (1) - Aansturen
   // Starten van Aanvoerband
   RUNG wire#powerrail
      Contact( "Systeem RUN" )
      { S7_Templates := "time_type := Time" } "Timer_Aanvoerband".TON(pt := "PLCMemory".Offset_Timers.Aanvoer_Start_Offset, et =>)
      Coil( "Aanvoerband_Tag1" )
   END_RUNG
   // the same network as SCL:
   "Timer_Aanvoerband".TON(IN := "Systeem RUN", PT := "PLCMemory".Offset_Timers.Aanvoer_Start_Offset);
   "Aanvoerband_Tag1" := "Timer_Aanvoerband".Q;
END_REGION

REGION Network 3: Aanvoerband (2) - Set Drive
   // Set drive Aanvoerband (Drive 1)
   RUNG wire#powerrail
      Contact( "Aanvoerband_Tag1" )
      S_Coil( "Drive_1_Auto" )
   END_RUNG
   // the same network as SCL:
   IF "Aanvoerband_Tag1" THEN "Drive_1_Auto" := TRUE; END_IF;
END_REGION

REGION Network 4: Aanvoerband (3) - Stoppen
   // Stoppen van de aanvoerband
   RUNG wire#powerrail
      I_Contact( "Systeem RUN" )
      { S7_Templates := "time_type := Time" } "Uitlooptimer_Aanvoerband".TON(pt := "PLCMemory".Offset_Timers.Aanvoer_Stop_Offset, et =>)
      Coil( "Aanvoerband_Tag2" )
   END_RUNG
   // the same network as SCL:
   "Uitlooptimer_Aanvoerband".TON(IN := NOT "Systeem RUN", PT := "PLCMemory".Offset_Timers.Aanvoer_Stop_Offset);
   "Aanvoerband_Tag2" := "Uitlooptimer_Aanvoerband".Q;
END_REGION

REGION Network 5: Aanvoerband (4) - Reset Drive
   // Reset van Drive Aanvoerband (Drive 1)
   RUNG wire#powerrail
      Contact( "Aanvoerband_Tag2" )
      R_Coil( "Drive_1_Auto" )
   END_RUNG
   // the same network as SCL:
   IF "Aanvoerband_Tag2" THEN "Drive_1_Auto" := FALSE; END_IF;
END_REGION

REGION Network 6: Aanvoerband (5) - Set Speed 1
   RUNG wire#powerrail
      Contact( "PLCMemory".SpeedSettingBand )
      Coil( "Drive 1 Speed 1" )
   END_RUNG
   // the same network as SCL:
   "Drive 1 Speed 1" := "PLCMemory".SpeedSettingBand;
END_REGION

REGION Network 7: Voorverdeelwals (1) - Start
   RUNG wire#powerrail
      Contact( "Systeem RUN" )
      Contact( "Sensor Op Band" )
      S_Coil( "Drive_3_Auto" )
   END_RUNG
   // the same network as SCL:
   IF "Systeem RUN" AND "Sensor Op Band" THEN "Drive_3_Auto" := TRUE; END_IF;
END_REGION

REGION Network 8: Voorverdeelwals (2) - Timer
   RUNG wire#powerrail
      Contact( "Sensor Op Band" )
      { S7_Templates := "time_type := Time" } "IEC_Timer_0DB_5".TOF(pt := T#1500ms, et =>)
      Coil( "Timer_Memory" )
   END_RUNG
   // the same network as SCL:
   "IEC_Timer_0DB_5".TOF(IN := "Sensor Op Band", PT := T#1500ms);
   "Timer_Memory" := "IEC_Timer_0DB_5".Q;
END_REGION

REGION Network 9: Voorverdeelwals (3) - Memory
   RUNG wire#powerrail
      Contact( "Timer_Memory" )
      S_Coil( "Sensor_op_band_memory" )
   END_RUNG
   // the same network as SCL:
   IF "Timer_Memory" THEN "Sensor_op_band_memory" := TRUE; END_IF;
END_REGION

REGION Network 10: Voorverdeelwals (4) - Delaying
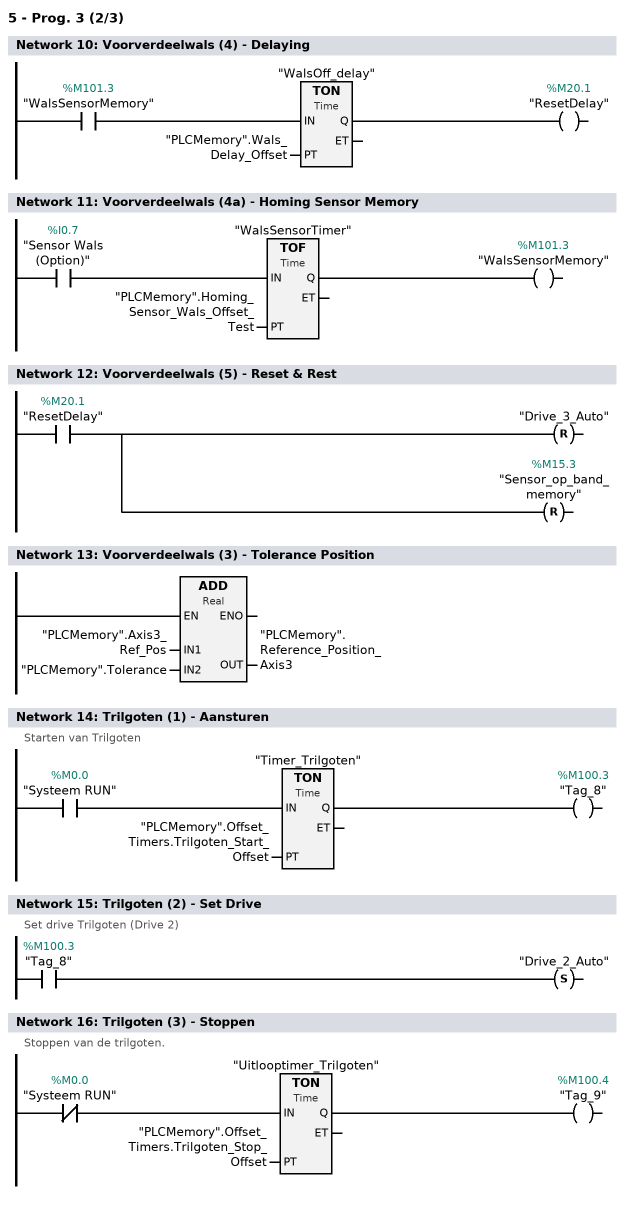
   RUNG wire#powerrail
      Contact( "WalsSensorMemory" )
      { S7_Templates := "time_type := Time" } "WalsOff_delay".TON(pt := "PLCMemory".Wals_Delay_Offset, et =>)
      Coil( "ResetDelay" )
   END_RUNG
   // the same network as SCL:
   "WalsOff_delay".TON(IN := "WalsSensorMemory", PT := "PLCMemory".Wals_Delay_Offset);
   "ResetDelay" := "WalsOff_delay".Q;
END_REGION

REGION Network 11: Voorverdeelwals (4a) - Homing Sensor Memory
   RUNG wire#powerrail
      Contact( "Sensor Wals (Option)" )
      { S7_Templates := "time_type := Time" } "WalsSensorTimer".TOF(pt := "PLCMemory".Homing_Sensor_Wals_Offset_Test, et =>)
      Coil( "WalsSensorMemory" )
   END_RUNG
   // the same network as SCL:
   "WalsSensorTimer".TOF(IN := "Sensor Wals (Option)", PT := "PLCMemory".Homing_Sensor_Wals_Offset_Test);
   "WalsSensorMemory" := "WalsSensorTimer".Q;
END_REGION

REGION Network 12: Voorverdeelwals (5) - Reset & Rest
   RUNG wire#powerrail
      Contact( "ResetDelay" )
      wire#w1
      R_Coil( "Drive_3_Auto" )
   END_RUNG
   RUNG wire#w1
      R_Coil( "Sensor_op_band_memory" )
   END_RUNG
   // the same network as SCL:
   IF "ResetDelay" THEN
       "Drive_3_Auto" := FALSE;
       "Sensor_op_band_memory" := FALSE;
   END_IF;
END_REGION

REGION Network 13: Voorverdeelwals (3) - Tolerance Position
   RUNG wire#powerrail
      { S7_Templates := "SrcType := Real"; S7_GenerateENO := "TRUE" } Add(in1 := "PLCMemory".Axis3_Ref_Pos, in2 := "PLCMemory".Tolerance, out => "PLCMemory".Reference_Position_Axis3)
   END_RUNG
   // the same network as SCL:
   "PLCMemory".Reference_Position_Axis3 := "PLCMemory".Axis3_Ref_Pos + "PLCMemory".Tolerance;
END_REGION

REGION Network 14: Trilgoten (1) - Aansturen
   // Starten van Trilgoten
   RUNG wire#powerrail
      Contact( "Systeem RUN" )
      { S7_Templates := "time_type := Time" } "Timer_Trilgoten".TON(pt := "PLCMemory".Offset_Timers.Trilgoten_Start_Offset, et =>)
      Coil( "Tag_8" )
   END_RUNG
   // the same network as SCL:
   "Timer_Trilgoten".TON(IN := "Systeem RUN", PT := "PLCMemory".Offset_Timers.Trilgoten_Start_Offset);
   "Tag_8" := "Timer_Trilgoten".Q;
END_REGION

REGION Network 15: Trilgoten (2) - Set Drive
   // Set drive Trilgoten (Drive 2)
   RUNG wire#powerrail
      Contact( "Tag_8" )
      S_Coil( "Drive_2_Auto" )
   END_RUNG
   // the same network as SCL:
   IF "Tag_8" THEN "Drive_2_Auto" := TRUE; END_IF;
END_REGION

REGION Network 16: Trilgoten (3) - Stoppen
   // Stoppen van de trilgoten.
   RUNG wire#powerrail
      I_Contact( "Systeem RUN" )
      { S7_Templates := "time_type := Time" } "Uitlooptimer_Trilgoten".TON(pt := "PLCMemory".Offset_Timers.Trilgoten_Stop_Offset, et =>)
      Coil( "Tag_9" )
   END_RUNG
   // the same network as SCL:
   "Uitlooptimer_Trilgoten".TON(IN := NOT "Systeem RUN", PT := "PLCMemory".Offset_Timers.Trilgoten_Stop_Offset);
   "Tag_9" := "Uitlooptimer_Trilgoten".Q;
END_REGION

REGION Network 17: Trilgoten (4) - Reset Drive
   // Reset van Drive Trilgoten (Drive 2)
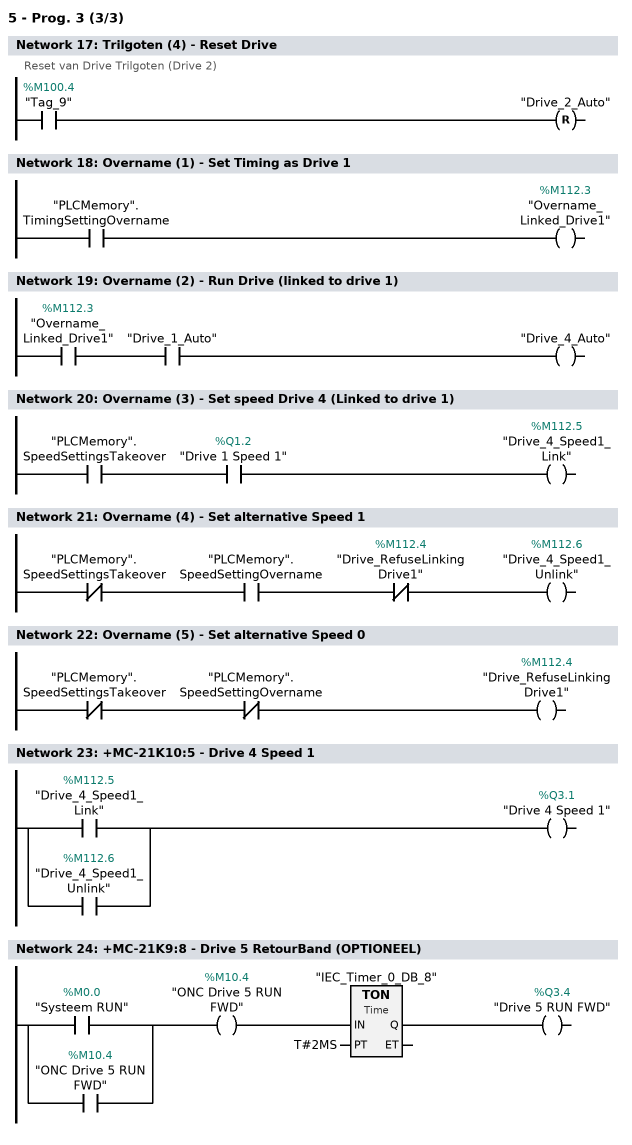
   RUNG wire#powerrail
      Contact( "Tag_9" )
      R_Coil( "Drive_2_Auto" )
   END_RUNG
   // the same network as SCL:
   IF "Tag_9" THEN "Drive_2_Auto" := FALSE; END_IF;
END_REGION

REGION Network 18: Overname (1) - Set Timing as Drive 1
   RUNG wire#powerrail
      Contact( "PLCMemory".TimingSettingOvername )
      Coil( "Overname_Linked_Drive1" )
   END_RUNG
   // the same network as SCL:
   "Overname_Linked_Drive1" := "PLCMemory".TimingSettingOvername;
END_REGION

REGION Network 19: Overname (2) - Run Drive (linked to drive 1)
   RUNG wire#powerrail
      Contact( "Overname_Linked_Drive1" )
      Contact( "Drive_1_Auto" )
      Coil( "Drive_4_Auto" )
   END_RUNG
   // the same network as SCL:
   "Drive_4_Auto" := "Overname_Linked_Drive1" AND "Drive_1_Auto";
END_REGION

REGION Network 20: Overname (3) - Set speed Drive 4 (Linked to drive 1)
   RUNG wire#powerrail
      Contact( "PLCMemory".SpeedSettingsTakeover )
      Contact( "Drive 1 Speed 1" )
      Coil( "Drive_4_Speed1_Link" )
   END_RUNG
   // the same network as SCL:
   "Drive_4_Speed1_Link" := "PLCMemory".SpeedSettingsTakeover AND "Drive 1 Speed 1";
END_REGION

REGION Network 21: Overname (4) - Set alternative Speed 1
   RUNG wire#powerrail
      I_Contact( "PLCMemory".SpeedSettingsTakeover )
      Contact( "PLCMemory".SpeedSettingOvername )
      I_Contact( "Drive_RefuseLinkingDrive1" )
      Coil( "Drive_4_Speed1_Unlink" )
   END_RUNG
   // the same network as SCL:
   "Drive_4_Speed1_Unlink" := NOT "PLCMemory".SpeedSettingsTakeover AND "PLCMemory".SpeedSettingOvername AND NOT "Drive_RefuseLinkingDrive1";
END_REGION

REGION Network 22: Overname (5) - Set alternative Speed 0
   RUNG wire#powerrail
      I_Contact( "PLCMemory".SpeedSettingsTakeover )
      I_Contact( "PLCMemory".SpeedSettingOvername )
      Coil( "Drive_RefuseLinkingDrive1" )
   END_RUNG
   // the same network as SCL:
   "Drive_RefuseLinkingDrive1" := NOT "PLCMemory".SpeedSettingsTakeover AND NOT "PLCMemory".SpeedSettingOvername;
END_REGION

REGION Network 23: +MC-21K10:5 - Drive 4 Speed 1
   RUNG wire#powerrail
      Contact( "Drive_4_Speed1_Link" )
      wire#w1
      Coil( "Drive 4 Speed 1" )
   END_RUNG
   RUNG wire#powerrail
      Contact( "Drive_4_Speed1_Unlink" )
   END_RUNG wire#w1
   // the same network as SCL:
   "Drive 4 Speed 1" := "Drive_4_Speed1_Link" OR "Drive_4_Speed1_Unlink";
END_REGION

REGION Network 24: +MC-21K9:8 - Drive 5 RetourBand (OPTIONEEL)
   RUNG wire#powerrail
      Contact( "Systeem RUN" )
      wire#w1
      Coil( "ONC Drive 5 RUN FWD" )
      { S7_Templates := "time_type := Time" } "IEC_Timer_0_DB_8".TON(pt := T#2MS, et =>)
      Coil( "Drive 5 RUN FWD" )
   END_RUNG
   RUNG wire#powerrail
      Contact( "ONC Drive 5 RUN FWD" )
   END_RUNG wire#w1
   // the same network as SCL:
   "ONC Drive 5 RUN FWD" := "Systeem RUN" OR "ONC Drive 5 RUN FWD";
   "IEC_Timer_0_DB_8".TON(IN := "ONC Drive 5 RUN FWD", PT := T#2MS);
   "Drive 5 RUN FWD" := "IEC_Timer_0_DB_8".Q;
END_REGION
END_FUNCTION

FUNCTION "1 - Outputs" : Void   // FC5, LAD
VERSION : 0.1
// This Function program is for operating the machine automatic and manual.
// stored: AutoNumber true, IsIECCheckEnabled false, UDAEnableTagReadback false
   VAR_TEMP
      Valve_2_Pulse : Bool;
      BlowOff_Activated : Bool;
      BlowOffManual : Bool;
      Pulse1 : Bool;
   END_VAR
   VAR_TEMP   // added for the SCL form of the ladder/FBD networks
      _w1 : Bool;
   END_VAR
BEGIN

REGION Network 1: Drive 1 - Control
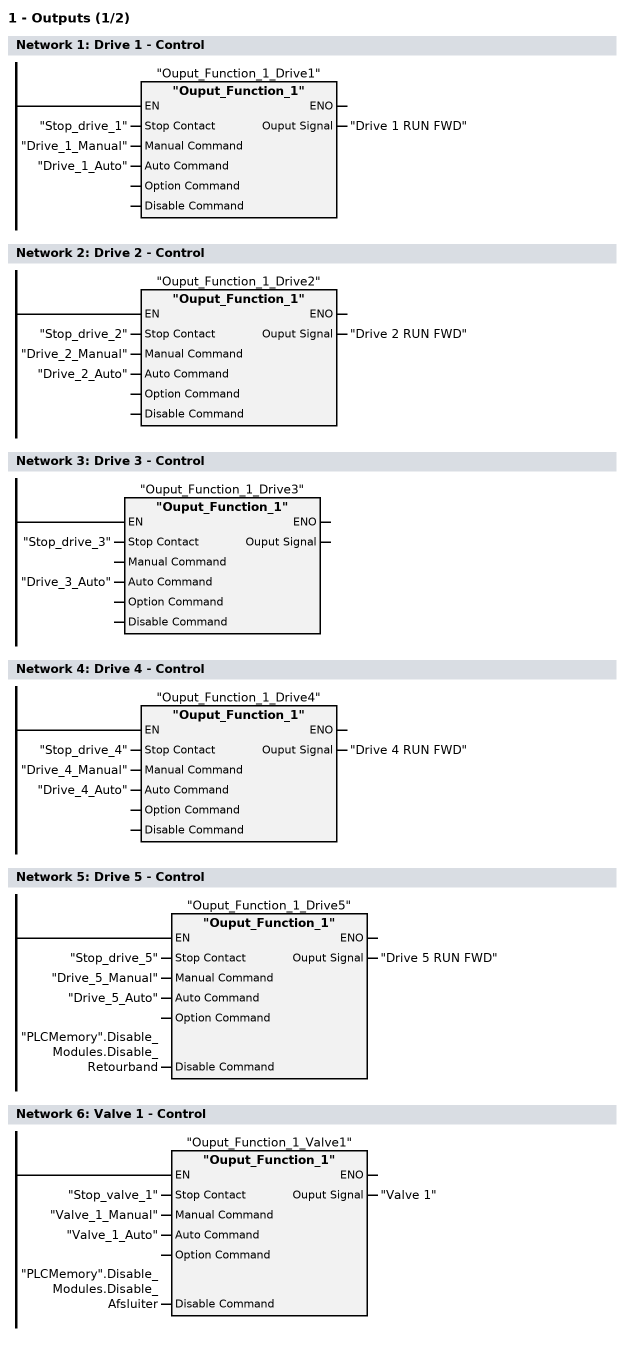
   RUNG wire#powerrail
      "Ouput_Function_1_Drive1"("Stop Contact" := "Stop_drive_1", "Manual Command" := "Drive_1_Manual", "Auto Command" := "Drive_1_Auto", "Option Command" :=, "Disable Command" :=, "Ouput Signal" => "Drive 1 RUN FWD")
   END_RUNG
   // the same network as SCL:
   "Ouput_Function_1_Drive1"("Stop Contact" := "Stop_drive_1",   // "Ouput_Function_1"
                           "Manual Command" := "Drive_1_Manual",
                           "Auto Command" := "Drive_1_Auto",
                           "Ouput Signal" => "Drive 1 RUN FWD");
END_REGION

REGION Network 2: Drive 2 - Control
   RUNG wire#powerrail
      "Ouput_Function_1_Drive2"("Stop Contact" := "Stop_drive_2", "Manual Command" := "Drive_2_Manual", "Auto Command" := "Drive_2_Auto", "Option Command" :=, "Disable Command" :=, "Ouput Signal" => "Drive 2 RUN FWD")
   END_RUNG
   // the same network as SCL:
   "Ouput_Function_1_Drive2"("Stop Contact" := "Stop_drive_2",   // "Ouput_Function_1"
                           "Manual Command" := "Drive_2_Manual",
                           "Auto Command" := "Drive_2_Auto",
                           "Ouput Signal" => "Drive 2 RUN FWD");
END_REGION

REGION Network 3: Drive 3 - Control
   RUNG wire#powerrail
      "Ouput_Function_1_Drive3"("Stop Contact" := "Stop_drive_3", "Manual Command" :=, "Auto Command" := "Drive_3_Auto", "Option Command" :=, "Disable Command" :=, "Ouput Signal" =>)
   END_RUNG
   // the same network as SCL:
   "Ouput_Function_1_Drive3"("Stop Contact" := "Stop_drive_3", "Auto Command" := "Drive_3_Auto");   // "Ouput_Function_1"
END_REGION

REGION Network 4: Drive 4 - Control
   RUNG wire#powerrail
      "Ouput_Function_1_Drive4"("Stop Contact" := "Stop_drive_4", "Manual Command" := "Drive_4_Manual", "Auto Command" := "Drive_4_Auto", "Option Command" :=, "Disable Command" :=, "Ouput Signal" => "Drive 4 RUN FWD")
   END_RUNG
   // the same network as SCL:
   "Ouput_Function_1_Drive4"("Stop Contact" := "Stop_drive_4",   // "Ouput_Function_1"
                           "Manual Command" := "Drive_4_Manual",
                           "Auto Command" := "Drive_4_Auto",
                           "Ouput Signal" => "Drive 4 RUN FWD");
END_REGION

REGION Network 5: Drive 5 - Control
   RUNG wire#powerrail
      "Ouput_Function_1_Drive5"("Stop Contact" := "Stop_drive_5", "Manual Command" := "Drive_5_Manual", "Auto Command" := "Drive_5_Auto", "Option Command" :=, "Disable Command" := "PLCMemory".Disable_Modules.Disable_Retourband, "Ouput Signal" => "Drive 5 RUN FWD")
   END_RUNG
   // the same network as SCL:
   "Ouput_Function_1_Drive5"("Stop Contact" := "Stop_drive_5",   // "Ouput_Function_1"
                           "Manual Command" := "Drive_5_Manual",
                           "Auto Command" := "Drive_5_Auto",
                           "Disable Command" := "PLCMemory".Disable_Modules.Disable_Retourband,
                           "Ouput Signal" => "Drive 5 RUN FWD");
END_REGION

REGION Network 6: Valve 1 - Control
   RUNG wire#powerrail
      "Ouput_Function_1_Valve1"("Stop Contact" := "Stop_valve_1", "Manual Command" := "Valve_1_Manual", "Auto Command" := "Valve_1_Auto", "Option Command" :=, "Disable Command" := "PLCMemory".Disable_Modules.Disable_Afsluiter, "Ouput Signal" => "Valve 1")
   END_RUNG
   // the same network as SCL:
   "Ouput_Function_1_Valve1"("Stop Contact" := "Stop_valve_1",   // "Ouput_Function_1"
                           "Manual Command" := "Valve_1_Manual",
                           "Auto Command" := "Valve_1_Auto",
                           "Disable Command" := "PLCMemory".Disable_Modules.Disable_Afsluiter,
                           "Ouput Signal" => "Valve 1");
END_REGION

REGION Network 7: Valve 2 - Control
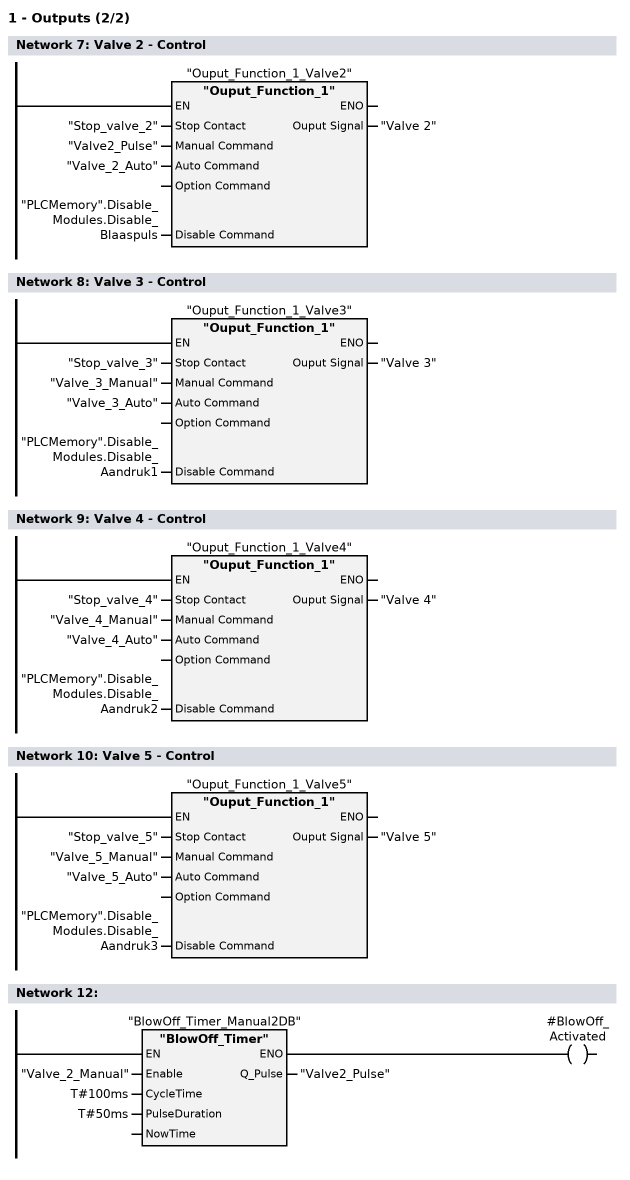
   RUNG wire#powerrail
      "Ouput_Function_1_Valve2"("Stop Contact" := "Stop_valve_2", "Manual Command" := "Valve2_Pulse", "Auto Command" := "Valve_2_Auto", "Option Command" :=, "Disable Command" := "PLCMemory".Disable_Modules.Disable_Blaaspuls, "Ouput Signal" => "Valve 2")
   END_RUNG
   // the same network as SCL:
   "Ouput_Function_1_Valve2"("Stop Contact" := "Stop_valve_2",   // "Ouput_Function_1"
                           "Manual Command" := "Valve2_Pulse",
                           "Auto Command" := "Valve_2_Auto",
                           "Disable Command" := "PLCMemory".Disable_Modules.Disable_Blaaspuls,
                           "Ouput Signal" => "Valve 2");
END_REGION

REGION Network 8: Valve 3 - Control
   RUNG wire#powerrail
      "Ouput_Function_1_Valve3"("Stop Contact" := "Stop_valve_3", "Manual Command" := "Valve_3_Manual", "Auto Command" := "Valve_3_Auto", "Option Command" :=, "Disable Command" := "PLCMemory".Disable_Modules.Disable_Aandruk1, "Ouput Signal" => "Valve 3")
   END_RUNG
   // the same network as SCL:
   "Ouput_Function_1_Valve3"("Stop Contact" := "Stop_valve_3",   // "Ouput_Function_1"
                           "Manual Command" := "Valve_3_Manual",
                           "Auto Command" := "Valve_3_Auto",
                           "Disable Command" := "PLCMemory".Disable_Modules.Disable_Aandruk1,
                           "Ouput Signal" => "Valve 3");
END_REGION

REGION Network 9: Valve 4 - Control
   RUNG wire#powerrail
      "Ouput_Function_1_Valve4"("Stop Contact" := "Stop_valve_4", "Manual Command" := "Valve_4_Manual", "Auto Command" := "Valve_4_Auto", "Option Command" :=, "Disable Command" := "PLCMemory".Disable_Modules.Disable_Aandruk2, "Ouput Signal" => "Valve 4")
   END_RUNG
   // the same network as SCL:
   "Ouput_Function_1_Valve4"("Stop Contact" := "Stop_valve_4",   // "Ouput_Function_1"
                           "Manual Command" := "Valve_4_Manual",
                           "Auto Command" := "Valve_4_Auto",
                           "Disable Command" := "PLCMemory".Disable_Modules.Disable_Aandruk2,
                           "Ouput Signal" => "Valve 4");
END_REGION

REGION Network 10: Valve 5 - Control
   RUNG wire#powerrail
      "Ouput_Function_1_Valve5"("Stop Contact" := "Stop_valve_5", "Manual Command" := "Valve_5_Manual", "Auto Command" := "Valve_5_Auto", "Option Command" :=, "Disable Command" := "PLCMemory".Disable_Modules.Disable_Aandruk3, "Ouput Signal" => "Valve 5")
   END_RUNG
   // the same network as SCL:
   "Ouput_Function_1_Valve5"("Stop Contact" := "Stop_valve_5",   // "Ouput_Function_1"
                           "Manual Command" := "Valve_5_Manual",
                           "Auto Command" := "Valve_5_Auto",
                           "Disable Command" := "PLCMemory".Disable_Modules.Disable_Aandruk3,
                           "Ouput Signal" => "Valve 5");
END_REGION

REGION Network 11: Blow Off Manual
END_REGION

REGION Network 12
   RUNG wire#powerrail
      "BlowOff_Timer_Manual2DB"(Enable := "Valve_2_Manual", CycleTime := T#100ms, PulseDuration := T#50ms, NowTime :=, Q_Pulse => "Valve2_Pulse")
      Coil( #BlowOff_Activated )
   END_RUNG
   // the same network as SCL:
   "BlowOff_Timer_Manual2DB"(Enable := "Valve_2_Manual",   // "BlowOff_Timer"
                           CycleTime := T#100ms,
                           PulseDuration := T#50ms,
                           Q_Pulse => "Valve2_Pulse",
                           ENO => #_w1);
   #BlowOff_Activated := #_w1;
END_REGION
END_FUNCTION

FUNCTION_BLOCK "Ouput_Function_1"   // FB8, FBD
TITLE = Ouput Controller Function Block
VERSION : 0.1
// stored: AutoNumber true, IsIECCheckEnabled false, UDAEnableTagReadback false
   VAR_INPUT
      "Stop Contact" : Bool;
      "Manual Command" : Bool;
      "Auto Command" : Bool;
      "Option Command" : Bool;
      "Disable Command" : Bool;
   END_VAR
   VAR_OUTPUT
      "Ouput Signal" : Bool;
   END_VAR
BEGIN

REGION Network 1: Ouput Controller
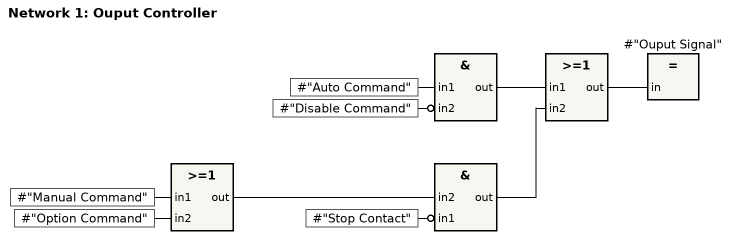
   #"Ouput Signal" := (#"Auto Command" AND NOT #"Disable Command") OR ((#"Manual Command" OR #"Option Command") AND NOT #"Stop Contact");
END_REGION
END_FUNCTION_BLOCK

FUNCTION "6 - Storingsmelding" : Void   // FC8, LAD
TITLE = Warnings
VERSION : 0.1
// This program block is for audible & visual warnings.
// stored: AutoNumber true, IsIECCheckEnabled false, UDAEnableTagReadback false
   VAR_TEMP
      "Wals Sensor Controlled" : Bool;
      "Infeed Sensor Controlled" : Bool;
   END_VAR
   VAR CONSTANT
      "Sensor 2 (option)" : Bool := TRUE;
   END_VAR
   VAR_TEMP   // added for the SCL form of the ladder/FBD networks
      _w1 : Bool;
   END_VAR
BEGIN

REGION Network 1: +MC-21K6:5 - Bel Storing
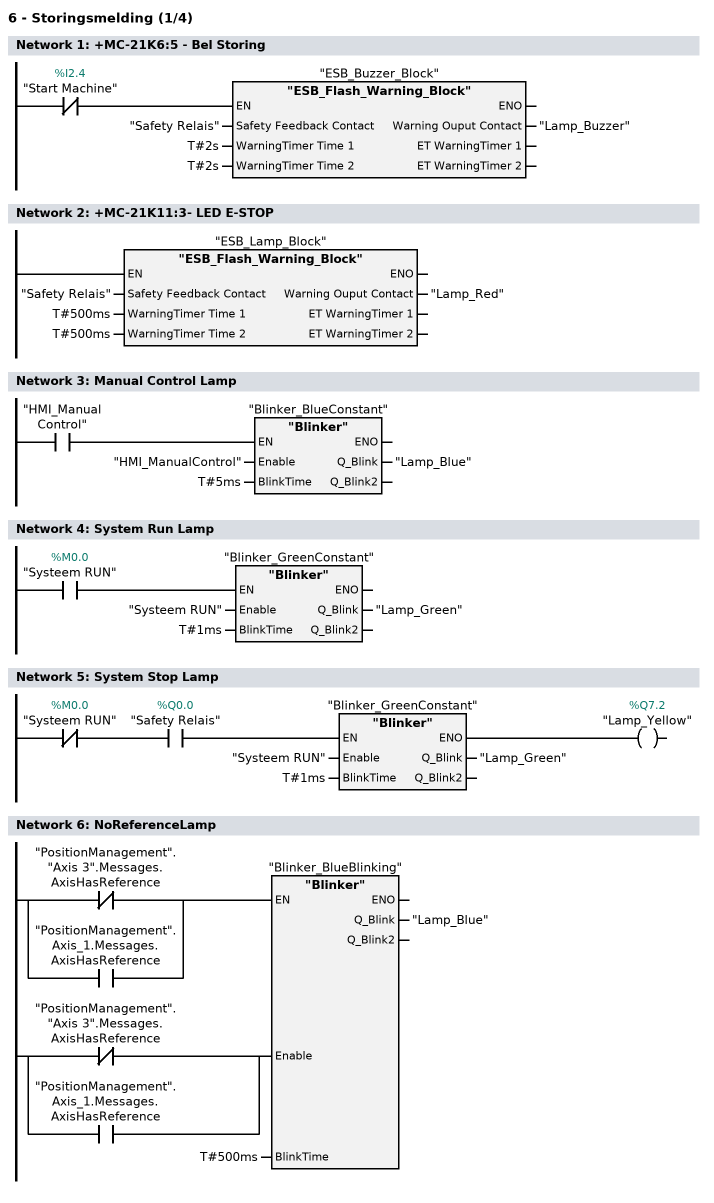
   RUNG wire#powerrail
      I_Contact( "Start Machine" )
      "ESB_Buzzer_Block"("Safety Feedback Contact" := "Safety Relais", "WarningTimer Time 1" := T#2s, "WarningTimer Time 2" := T#2s, "Warning Ouput Contact" => "Lamp_Buzzer", "ET WarningTimer 1" =>, "ET WarningTimer 2" =>)
   END_RUNG
   // the same network as SCL:
   IF NOT "Start Machine" THEN
       "ESB_Buzzer_Block"("Safety Feedback Contact" := "Safety Relais",   // "ESB_Flash_Warning_Block"
                          "WarningTimer Time 1" := T#2s,
                          "WarningTimer Time 2" := T#2s,
                          "Warning Ouput Contact" => "Lamp_Buzzer");
   END_IF;
END_REGION

REGION Network 2: +MC-21K11:3- LED E-STOP
   RUNG wire#powerrail
      "ESB_Lamp_Block"("Safety Feedback Contact" := "Safety Relais", "WarningTimer Time 1" := T#500ms, "WarningTimer Time 2" := T#500ms, "Warning Ouput Contact" => "Lamp_Red", "ET WarningTimer 1" =>, "ET WarningTimer 2" =>)
   END_RUNG
   // the same network as SCL:
   "ESB_Lamp_Block"("Safety Feedback Contact" := "Safety Relais",   // "ESB_Flash_Warning_Block"
                    "WarningTimer Time 1" := T#500ms,
                    "WarningTimer Time 2" := T#500ms,
                    "Warning Ouput Contact" => "Lamp_Red");
END_REGION

REGION Network 3: Manual Control Lamp
   RUNG wire#powerrail
      Contact( "HMI_ManualControl" )
      "Blinker_BlueConstant"(Enable := "HMI_ManualControl", BlinkTime := T#5ms, Q_Blink => "Lamp_Blue", Q_Blink2 =>)
   END_RUNG
   // the same network as SCL:
   IF "HMI_ManualControl" THEN
       "Blinker_BlueConstant"(Enable := "HMI_ManualControl", BlinkTime := T#5ms, Q_Blink => "Lamp_Blue");   // "Blinker"
   END_IF;
END_REGION

REGION Network 4: System Run Lamp
   RUNG wire#powerrail
      Contact( "Systeem RUN" )
      "Blinker_GreenConstant"(Enable := "Systeem RUN", BlinkTime := T#1ms, Q_Blink => "Lamp_Green", Q_Blink2 =>)
   END_RUNG
   // the same network as SCL:
   IF "Systeem RUN" THEN
       "Blinker_GreenConstant"(Enable := "Systeem RUN", BlinkTime := T#1ms, Q_Blink => "Lamp_Green");   // "Blinker"
   END_IF;
END_REGION

REGION Network 5: System Stop Lamp
   RUNG wire#powerrail
      I_Contact( "Systeem RUN" )
      Contact( "Safety Relais" )
      "Blinker_GreenConstant"(Enable := "Systeem RUN", BlinkTime := T#1ms, Q_Blink => "Lamp_Green", Q_Blink2 =>)
      Coil( "Lamp_Yellow" )
   END_RUNG
   // the same network as SCL:
   "Blinker_GreenConstant"(EN := NOT "Systeem RUN" AND "Safety Relais",   // "Blinker"
                           Enable := "Systeem RUN",
                           BlinkTime := T#1ms,
                           Q_Blink => "Lamp_Green",
                           ENO => #_w1);
   "Lamp_Yellow" := #_w1;
END_REGION

REGION Network 6: NoReferenceLamp
   RUNG wire#powerrail
      I_Contact( "PositionManagement"."Axis 3".Messages.AxisHasReference )
      wire#w1
      "Blinker_BlueBlinking"(Enable := wire#w2, BlinkTime := T#500ms, Q_Blink => "Lamp_Blue", Q_Blink2 =>)
   END_RUNG
   RUNG wire#powerrail
      Contact( "PositionManagement".Axis_1.Messages.AxisHasReference )
   END_RUNG wire#w1
   RUNG wire#powerrail
      I_Contact( "PositionManagement"."Axis 3".Messages.AxisHasReference )
   END_RUNG wire#w2
   RUNG wire#powerrail
      Contact( "PositionManagement".Axis_1.Messages.AxisHasReference )
   END_RUNG wire#w2
   // the same network as SCL:
   IF NOT "PositionManagement"."Axis 3".Messages.AxisHasReference OR "PositionManagement".Axis_1.Messages.AxisHasReference THEN
       "Blinker_BlueBlinking"(Enable := NOT "PositionManagement"."Axis 3".Messages.AxisHasReference OR "PositionManagement".Axis_1.Messages.AxisHasReference,   // "Blinker"
                              BlinkTime := T#500ms,
                              Q_Blink => "Lamp_Blue");
   END_IF;
END_REGION

REGION Network 7: Fill Trechter Delay Function
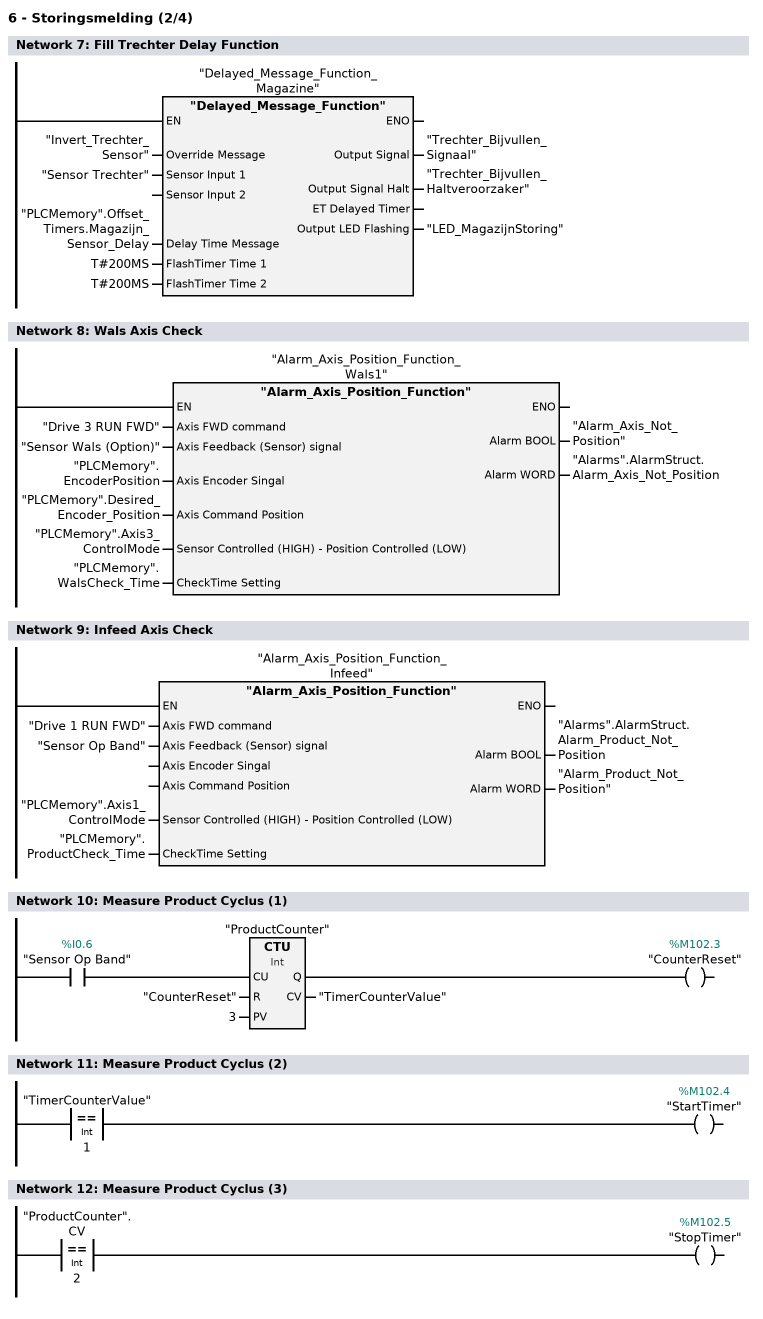
   RUNG wire#powerrail
      "Delayed_Message_Function_Magazine"("Override Message" := "Invert_Trechter_Sensor", "Sensor Input 1" := "Sensor Trechter", "Sensor Input 2" :=, "Delay Time Message" := "PLCMemory".Offset_Timers.Magazijn_Sensor_Delay, "FlashTimer Time 1" := T#200MS, "FlashTimer Time 2" := T#200MS, "Output Signal" => "Trechter_Bijvullen_Signaal", "Output Signal Halt" => "Trechter_Bijvullen_Haltveroorzaker", "ET Delayed Timer" =>, "Output LED Flashing" => "LED_MagazijnStoring")
   END_RUNG
   // the same network as SCL:
   "Delayed_Message_Function_Magazine"("Override Message" := "Invert_Trechter_Sensor",   // "Delayed_Message_Function"
                           "Sensor Input 1" := "Sensor Trechter",
                           "Delay Time Message" := "PLCMemory".Offset_Timers.Magazijn_Sensor_Delay,
                           "FlashTimer Time 1" := T#200MS,
                           "FlashTimer Time 2" := T#200MS,
                           "Output Signal" => "Trechter_Bijvullen_Signaal",
                           "Output Signal Halt" => "Trechter_Bijvullen_Haltveroorzaker",
                           "Output LED Flashing" => "LED_MagazijnStoring");
END_REGION

REGION Network 8: Wals Axis Check
   RUNG wire#powerrail
      "Alarm_Axis_Position_Function_Wals1"("Axis FWD command" := "Drive 3 RUN FWD", "Axis Feedback (Sensor) signal" := "Sensor Wals (Option)", "Axis Encoder Singal" := "PLCMemory".EncoderPosition, "Axis Command Position" := "PLCMemory".Desired_Encoder_Position, "Sensor Controlled (HIGH) - Position Controlled (LOW)" := "PLCMemory".Axis3_ControlMode, "CheckTime Setting" := "PLCMemory".WalsCheck_Time, "Alarm BOOL" => "Alarm_Axis_Not_Position", "Alarm WORD" => "Alarms".AlarmStruct.Alarm_Axis_Not_Position)
   END_RUNG
   // the same network as SCL:
   "Alarm_Axis_Position_Function_Wals1"("Axis FWD command" := "Drive 3 RUN FWD",   // "Alarm_Axis_Position_Function"
                           "Axis Feedback (Sensor) signal" := "Sensor Wals (Option)",
                           "Axis Encoder Singal" := "PLCMemory".EncoderPosition,
                           "Axis Command Position" := "PLCMemory".Desired_Encoder_Position,
                           "Sensor Controlled (HIGH) - Position Controlled (LOW)" := "PLCMemory".Axis3_ControlMode,
                           "CheckTime Setting" := "PLCMemory".WalsCheck_Time,
                           "Alarm BOOL" => "Alarm_Axis_Not_Position",
                           "Alarm WORD" => "Alarms".AlarmStruct.Alarm_Axis_Not_Position);
END_REGION

REGION Network 9: Infeed Axis Check
   RUNG wire#powerrail
      "Alarm_Axis_Position_Function_Infeed"("Axis FWD command" := "Drive 1 RUN FWD", "Axis Feedback (Sensor) signal" := "Sensor Op Band", "Axis Encoder Singal" :=, "Axis Command Position" :=, "Sensor Controlled (HIGH) - Position Controlled (LOW)" := "PLCMemory".Axis1_ControlMode, "CheckTime Setting" := "PLCMemory".ProductCheck_Time, "Alarm BOOL" => "Alarms".AlarmStruct.Alarm_Product_Not_Position, "Alarm WORD" => "Alarm_Product_Not_Position")
   END_RUNG
   // the same network as SCL:
   "Alarm_Axis_Position_Function_Infeed"("Axis FWD command" := "Drive 1 RUN FWD",   // "Alarm_Axis_Position_Function"
                           "Axis Feedback (Sensor) signal" := "Sensor Op Band",
                           "Sensor Controlled (HIGH) - Position Controlled (LOW)" := "PLCMemory".Axis1_ControlMode,
                           "CheckTime Setting" := "PLCMemory".ProductCheck_Time,
                           "Alarm BOOL" => "Alarms".AlarmStruct.Alarm_Product_Not_Position,
                           "Alarm WORD" => "Alarm_Product_Not_Position");
END_REGION

REGION Network 10: Measure Product Cyclus (1)
   RUNG wire#powerrail
      Contact( "Sensor Op Band" )
      { S7_Templates := "value_type := Int" } "ProductCounter".CTU(r := "CounterReset", pv := 3, cv => "TimerCounterValue")
      Coil( "CounterReset" )
   END_RUNG
   // the same network as SCL:
   "ProductCounter".CTU(CU := "Sensor Op Band", R := "CounterReset", PV := 3, CV => "TimerCounterValue");
   "CounterReset" := "ProductCounter".Q;
END_REGION

REGION Network 11: Measure Product Cyclus (2)
   RUNG wire#powerrail
      { S7_Templates := "SrcType := Int" } EQ_Contact(in1 := "TimerCounterValue", in2 := 1)
      Coil( "StartTimer" )
   END_RUNG
   // the same network as SCL:
   "StartTimer" := "TimerCounterValue" = 1;
END_REGION

REGION Network 12: Measure Product Cyclus (3)
   RUNG wire#powerrail
      { S7_Templates := "SrcType := Int" } EQ_Contact(in1 := "ProductCounter".CV, in2 := 2)
      Coil( "StopTimer" )
   END_RUNG
   // the same network as SCL:
   "StopTimer" := "ProductCounter".CV = 2;
END_REGION

REGION Network 13: Measure Product Cyclus (4)
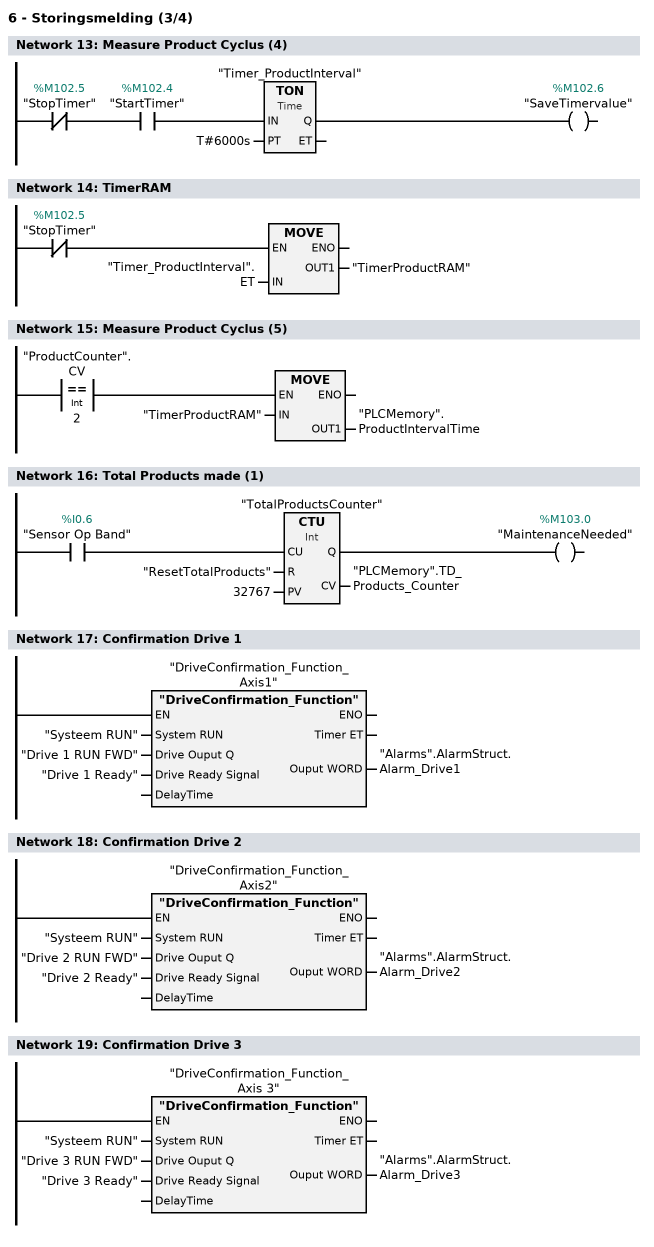
   RUNG wire#powerrail
      I_Contact( "StopTimer" )
      Contact( "StartTimer" )
      { S7_Templates := "time_type := Time" } "Timer_ProductInterval".TON(pt := T#6000s, et =>)
      Coil( "SaveTimervalue" )
   END_RUNG
   // the same network as SCL:
   "Timer_ProductInterval".TON(IN := NOT "StopTimer" AND "StartTimer", PT := T#6000s);
   "SaveTimervalue" := "Timer_ProductInterval".Q;
END_REGION

REGION Network 14: TimerRAM
   RUNG wire#powerrail
      I_Contact( "StopTimer" )
      { S7_GenerateENO := "TRUE" } Move(in := "Timer_ProductInterval".ET, out1 => "TimerProductRAM")
   END_RUNG
   // the same network as SCL:
   IF NOT "StopTimer" THEN "TimerProductRAM" := "Timer_ProductInterval".ET; END_IF;
END_REGION

REGION Network 15: Measure Product Cyclus (5)
   RUNG wire#powerrail
      { S7_Templates := "SrcType := Int" } EQ_Contact(in1 := "ProductCounter".CV, in2 := 2)
      { S7_GenerateENO := "TRUE" } Move(in := "TimerProductRAM", out1 => "PLCMemory".ProductIntervalTime)
   END_RUNG
   // the same network as SCL:
   IF "ProductCounter".CV = 2 THEN "PLCMemory".ProductIntervalTime := "TimerProductRAM"; END_IF;
END_REGION

